LIN {X 0,Y 488.78,Z 301.595,A -85,B 0,C 180,E1 22660.647,E2 22660.647} C_VEL
LIN {X 0,Y 488.836,Z 301.585,A -85,B 0,C 180,E1 22657.258,E2 22657.258} C_VEL
LIN {X 0,Y 488.792,Z 301.599,A -85,B 0,C 180,E1 22653.779,E2 22653.779} C_VEL
LIN {X 0,Y 488.782,Z 301.597,A -85,B 0,C 180,E1 22650.328,E2 22650.328} C_VEL
LIN {X 0,Y 488.822,Z 301.594,A -85,B 0,C 180,E1 22646.898,E2 22646.898} C_VEL
LIN {X 0,Y 488.826,Z 301.564,A -85,B 0,C 180,E1 22643.301,E2 22643.301} C_VEL
LIN {X 0,Y 488.793,Z 301.59,A -85,B 0,C 180,E1 22639.883,E2 22639.883} C_VEL
LIN {X 0,Y 488.796,Z 301.598,A -85,B 0,C 180,E1 22636.225,E2 22636.225} C_VEL
LIN {X 0,Y 488.826,Z 301.575,A -85,B 0,C 180,E1 22632.751,E2 22632.751} C_VEL
LIN {X 0,Y 488.839,Z 301.65,A -85,B 0,C 180,E1 22631.1,E2 22631.1} C_VEL
LIN {X 0,Y 489.193,Z 303.151,A -85,B 0,C 180,E1 22630.866,E2 22630.866} C_VEL
LIN {X 0,Y 497.247,Z 321.838,A -85,B 0,C 180,E1 22628.815,E2 22628.815} C_VEL
LIN {X 0,Y 502.538,Z 335.639,A -85,B 0,C 180,E1 22627.431,E2 22627.431} C_VEL
LIN {X 0,Y 500.242,Z 388.267,A -85,B 0,C 180,E1 22624.007,E2 22624.007} C_VEL
LIN {X 0,Y 502.743,Z 409.204,A -85,B 0,C 180,E1 22623.487,E2 22623.487} C_VEL
LIN {X 0,Y 499.827,Z 627.706,A -85,B 0,C 180,E1 22620.075,E2 22620.075} C_VEL
LIN {X 0,Y 499.277,Z 655.552,A -85,B 0,C 180,E1 22619.579,E2 22619.579} C_VEL
LIN {X 0,Y 498.434,Z 677.22,A -85,B 0,C 180,E1 22618.977,E2 22618.977} C_VEL
LIN {X 0,Y 497.483,Z 697.861,A -85,B 0,C 180,E1 22618.184,E2 22618.184} C_VEL
LIN {X 0,Y 496.413,Z 717.588,A -85,B 0,C 180,E1 22617.207,E2 22617.207} C_VEL
LIN {X 0,Y 495.194,Z 737.474,A -85,B 0,C 180,E1 22615.985,E2 22615.985} C_VEL
LIN {X 0,Y 493.989,Z 756.462,A -85,B 0,C 180,E1 22614.565,E2 22614.565} C_VEL
LIN {X 0,Y 492.797,Z 774.049,A -85,B 0,C 180,E1 22612.989,E2 22612.989} C_VEL
LIN {X 0,Y 491.739,Z 789.65,A -85,B 0,C 180,E1 22611.343,E2 22611.343} C_VEL
LIN {X 0,Y 490.759,Z 804.438,A -85,B 0,C 180,E1 22609.519,E2 22609.519} C_VEL
LIN {X 0,Y 490.048,Z 815.118,A -85,B 0,C 180,E1 22607.944,E2 22607.944} C_VEL
LIN {X 0,Y 489.28,Z 826.646,A -85,B 0,C 180,E1 22605.892,E2 22605.892} C_VEL
LIN {X 0,Y 488.709,Z 836.846,A -85,B 0,C 180,E1 22603.728,E2 22603.728} C_VEL
LIN {X 0,Y 488.31,Z 845.655,A -85,B 0,C 180,E1 22601.456,E2 22601.456} C_VEL
LIN {X 0,Y 488.088,Z 852.685,A -85,B 0,C 180,E1 22599.194,E2 22599.194} C_VEL
LIN {X 0,Y 487.97,Z 858.26,A -85,B 0,C 180,E1 22596.825,E2 22596.825} C_VEL
LIN {X 0,Y 487.913,Z 862.087,A -85,B 0,C 180,E1 22594.466,E2 22594.466} C_VEL
LIN {X 0,Y 487.908,Z 864.304,A -85,B 0,C 180,E1 22592.114,E2 22592.114} C_VEL
LIN {X 0,Y 487.906,Z 864.962,A -85,B 0,C 180,E1 22589.765,E2 22589.765} C_VEL
LIN {X 0,Y 487.905,Z 864.03,A -85,B 0,C 180,E1 22587.416,E2 22587.416} C_VEL
LIN {X 0,Y 487.929,Z 861.446,A -85,B 0,C 180,E1 22585.063,E2 22585.063} C_VEL
LIN {X 0,Y 487.987,Z 857.244,A -85,B 0,C 180,E1 22582.702,E2 22582.702} C_VEL
LIN {X 0,Y 488.126,Z 851.326,A -85,B 0,C 180,E1 22580.331,E2 22580.331} C_VEL
LIN {X 0,Y 488.381,Z 844.01,A -85,B 0,C 180,E1 22578.067,E2 22578.067} C_VEL
LIN {X 0,Y 488.823,Z 834.789,A -85,B 0,C 180,E1 22575.792,E2 22575.792} C_VEL
LIN {X 0,Y 489.44,Z 824.106,A -85,B 0,C 180,E1 22573.626,E2 22573.626} C_VEL
LIN {X 0,Y 490.253,Z 812.019,A -85,B 0,C 180,E1 22571.572,E2 22571.572} C_VEL
LIN {X 0,Y 491.025,Z 800.468,A -85,B 0,C 180,E1 22569.954,E2 22569.954} C_VEL
LIN {X 0,Y 492.085,Z 784.784,A -85,B 0,C 180,E1 22568.109,E2 22568.109} C_VEL
LIN {X 0,Y 493.241,Z 767.415,A -85,B 0,C 180,E1 22566.385,E2 22566.385} C_VEL
LIN {X 0,Y 494.4,Z 750.145,A -85,B 0,C 180,E1 22564.94,E2 22564.94} C_VEL
LIN {X 0,Y 495.552,Z 731.825,A -85,B 0,C 180,E1 22563.649,E2 22563.649} C_VEL
LIN {X 0,Y 496.728,Z 711.811,A -85,B 0,C 180,E1 22562.487,E2 22562.487} C_VEL
LIN {X 0,Y 497.765,Z 692.146,A -85,B 0,C 180,E1 22561.572,E2 22561.572} C_VEL
LIN {X 0,Y 498.696,Z 671.504,A -85,B 0,C 180,E1 22560.837,E2 22560.837} C_VEL
LIN {X 0,Y 499.453,Z 649.882,A -85,B 0,C 180,E1 22560.293,E2 22560.293} C_VEL
LIN {X 0,Y 502.656,Z 414.695,A -85,B 0,C 180,E1 22556.6,E2 22556.6} C_VEL
LIN {X 0,Y 502.523,Z 405.875,A -85,B 0,C 180,E1 22556.443,E2 22556.443} C_VEL
LIN {X 0,Y 500.189,Z 387.515,A -85,B 0,C 180,E1 22555.965,E2 22555.965} C_VEL
LIN {X 0,Y 502.552,Z 335.273,A -85,B 0,C 180,E1 22552.545,E2 22552.545} C_VEL
LIN {X 0,Y 494.184,Z 314.542,A -85,B 0,C 180,E1 22550.409,E2 22550.409} C_VEL
LIN {X 0,Y 488.897,Z 302.02,A -85,B 0,C 180,E1 22548.995,E2 22548.995} C_VEL
LIN {X 0,Y 488.827,Z 301.588,A -85,B 0,C 180,E1 22548.648,E2 22548.648} C_VEL
LIN {X 0,Y 488.832,Z 301.584,A -85,B 0,C 180,E1 22545.049,E2 22545.049} C_VEL
LIN {X 0,Y 488.802,Z 301.566,A -85,B 0,C 180,E1 22541.51,E2 22541.51} C_VEL
LIN {X 0,Y 488.79,Z 301.592,A -85,B 0,C 180,E1 22538.004,E2 22538.004} C_VEL
LIN {X 0,Y 488.813,Z 301.58,A -85,B 0,C 180,E1 22534.482,E2 22534.482} C_VEL
LIN {X 0,Y 488.834,Z 301.587,A -85,B 0,C 180,E1 22530.89,E2 22530.89} C_VEL
LIN {X 0,Y 488.79,Z 301.591,A -85,B 0,C 180,E1 22527.403,E2 22527.403} C_VEL
LIN {X 0,Y 488.779,Z 301.593,A -85,B 0,C 180,E1 22523.884,E2 22523.884} C_VEL
LIN {X 0,Y 488.816,Z 301.598,A -85,B 0,C 180,E1 22520.473,E2 22520.473} C_VEL
LIN {X 0,Y 488.801,Z 301.592,A -85,B 0,C 180,E1 22517.008,E2 22517.008} C_VEL
LIN {X 0,Y 488.765,Z 301.585,A -85,B 0,C 180,E1 22513.606,E2 22513.606} C_VEL
LIN {X 0,Y 488.783,Z 301.596,A -85,B 0,C 180,E1 22510.132,E2 22510.132} C_VEL
LIN {X 0,Y 488.827,Z 301.591,A -85,B 0,C 180,E1 22506.577,E2 22506.577} C_VEL
LIN {X 0,Y 488.77,Z 301.59,A -85,B 0,C 180,E1 22503.049,E2 22503.049} C_VEL
LIN {X 0,Y 488.753,Z 301.6,A -85,B 0,C 180,E1 22499.648,E2 22499.648} C_VEL
LIN {X 0,Y 488.794,Z 301.59,A -85,B 0,C 180,E1 22496.247,E2 22496.247} C_VEL
LIN {X 0,Y 488.783,Z 301.599,A -85,B 0,C 180,E1 22492.79,E2 22492.79} C_VEL
LIN {X 0,Y 488.756,Z 301.598,A -85,B 0,C 180,E1 22489.39,E2 22489.39} C_VEL
LIN {X 0,Y 488.783,Z 301.585,A -85,B 0,C 180,E1 22485.911,E2 22485.911} C_VEL
LIN {X 0,Y 488.808,Z 301.6,A -85,B 0,C 180,E1 22482.501,E2 22482.501} C_VEL
LIN {X 0,Y 488.771,Z 301.593,A -85,B 0,C 180,E1 22479.023,E2 22479.023} C_VEL
LIN {X 0,Y 488.775,Z 301.586,A -85,B 0,C 180,E1 22475.464,E2 22475.464} C_VEL
LIN {X 0,Y 488.83,Z 301.592,A -85,B 0,C 180,E1 22472.069,E2 22472.069} C_VEL
LIN {X 0,Y 488.806,Z 301.597,A -85,B 0,C 180,E1 22468.534,E2 22468.534} C_VEL
LIN {X 0,Y 488.781,Z 301.595,A -85,B 0,C 180,E1 22465.056,E2 22465.056} C_VEL
LIN {X 0,Y 488.801,Z 301.594,A -85,B 0,C 180,E1 22461.549,E2 22461.549} C_VEL
LIN {X 0,Y 488.832,Z 301.59,A -85,B 0,C 180,E1 22458.022,E2 22458.022} C_VEL
LIN {X 0,Y 488.81,Z 301.571,A -85,B 0,C 180,E1 22454.448,E2 22454.448} C_VEL
LIN {X 0,Y 488.793,Z 301.6,A -85,B 0,C 180,E1 22450.887,E2 22450.887} C_VEL
LIN {X 0,Y 488.804,Z 301.585,A -85,B 0,C 180,E1 22447.277,E2 22447.277} C_VEL
LIN {X 0,Y 488.829,Z 301.571,A -85,B 0,C 180,E1 22443.803,E2 22443.803} C_VEL
LIN {X 0,Y 488.825,Z 301.575,A -85,B 0,C 180,E1 22443.535,E2 22443.535} C_VEL
LIN {X 0,Y 488.707,Z 302.659,A -85,B 0,C 180,E1 22443.028,E2 22443.028} C_VEL
LIN {X 0,Y 488.366,Z 306.029,A -85,B 0,C 180,E1 22442.479,E2 22442.479} C_VEL
LIN {X 0,Y 487.643,Z 319.511,A -85,B 0,C 180,E1 22441.022,E2 22441.022} C_VEL
LIN {X 0,Y 488.549,Z 324.711,A -85,B 0,C 180,E1 22440.361,E2 22440.361} C_VEL
LIN {X 0,Y 490.865,Z 331.872,A -85,B 0,C 180,E1 22439.399,E2 22439.399} C_VEL
LIN {X 0,Y 490.606,Z 339.583,A -85,B 0,C 180,E1 22438.658,E2 22438.658} C_VEL
LIN {X 0,Y 494.065,Z 356.306,A -85,B 0,C 180,E1 22438.141,E2 22438.141} C_VEL
LIN {X 0,Y 492.291,Z 551.901,A -85,B 0,C 180,E1 22435.29,E2 22435.29} C_VEL
LIN {X 0,Y 491.896,Z 570.892,A -85,B 0,C 180,E1 22434.786,E2 22434.786} C_VEL
LIN {X 0,Y 491.192,Z 588.904,A -85,B 0,C 180,E1 22434.087,E2 22434.087} C_VEL
LIN {X 0,Y 490.248,Z 606.351,A -85,B 0,C 180,E1 22433.179,E2 22433.179} C_VEL
LIN {X 0,Y 489.098,Z 622.756,A -85,B 0,C 180,E1 22432.095,E2 22432.095} C_VEL
LIN {X 0,Y 487.851,Z 638.101,A -85,B 0,C 180,E1 22430.839,E2 22430.839} C_VEL
LIN {X 0,Y 486.5,Z 652.717,A -85,B 0,C 180,E1 22429.379,E2 22429.379} C_VEL
LIN {X 0,Y 485.184,Z 666.107,A -85,B 0,C 180,E1 22427.757,E2 22427.757} C_VEL
LIN {X 0,Y 483.924,Z 678.429,A -85,B 0,C 180,E1 22425.949,E2 22425.949} C_VEL
LIN {X 0,Y 482.864,Z 689.222,A -85,B 0,C 180,E1 22424.02,E2 22424.02} C_VEL
LIN {X 0,Y 481.974,Z 698.544,A -85,B 0,C 180,E1 22421.973,E2 22421.973} C_VEL
LIN {X 0,Y 481.314,Z 706.381,A -85,B 0,C 180,E1 22419.807,E2 22419.807} C_VEL
LIN {X 0,Y 480.863,Z 712.699,A -85,B 0,C 180,E1 22417.527,E2 22417.527} C_VEL
LIN {X 0,Y 480.577,Z 717.234,A -85,B 0,C 180,E1 22415.252,E2 22415.252} C_VEL
LIN {X 0,Y 480.428,Z 720.208,A -85,B 0,C 180,E1 22412.863,E2 22412.863} C_VEL
LIN {X 0,Y 480.381,Z 721.437,A -85,B 0,C 180,E1 22410.477,E2 22410.477} C_VEL
LIN {X 0,Y 480.403,Z 720.959,A -85,B 0,C 180,E1 22408.092,E2 22408.092} C_VEL
LIN {X 0,Y 480.492,Z 718.906,A -85,B 0,C 180,E1 22405.824,E2 22405.824} C_VEL
LIN {X 0,Y 480.694,Z 715.237,A -85,B 0,C 180,E1 22403.551,E2 22403.551} C_VEL
LIN {X 0,Y 481.06,Z 709.851,A -85,B 0,C 180,E1 22401.273,E2 22401.273} C_VEL
LIN {X 0,Y 481.58,Z 703.016,A -85,B 0,C 180,E1 22399.11,E2 22399.11} C_VEL
LIN {X 0,Y 482.32,Z 694.791,A -85,B 0,C 180,E1 22397.063,E2 22397.063} C_VEL
LIN {X 0,Y 483.286,Z 684.793,A -85,B 0,C 180,E1 22395.054,E2 22395.054} C_VEL
LIN {X 0,Y 484.416,Z 673.543,A -85,B 0,C 180,E1 22393.204,E2 22393.204} C_VEL
LIN {X 0,Y 485.68,Z 661.12,A -85,B 0,C 180,E1 22391.517,E2 22391.517} C_VEL
LIN {X 0,Y 487.013,Z 647.199,A -85,B 0,C 180,E1 22389.95,E2 22389.95} C_VEL
LIN {X 0,Y 488.338,Z 632.237,A -85,B 0,C 180,E1 22388.564,E2 22388.564} C_VEL
LIN {X 0,Y 489.56,Z 616.352,A -85,B 0,C 180,E1 22387.364,E2 22387.364} C_VEL
LIN {X 0,Y 490.6,Z 600.329,A -85,B 0,C 180,E1 22386.393,E2 22386.393} C_VEL
LIN {X 0,Y 491.444,Z 583.063,A -85,B 0,C 180,E1 22385.575,E2 22385.575} C_VEL
LIN {X 0,Y 492.049,Z 564.71,A -85,B 0,C 180,E1 22384.938,E2 22384.938} C_VEL
LIN {X 0,Y 492.337,Z 545.999,A -85,B 0,C 180,E1 22384.513,E2 22384.513} C_VEL
LIN {X 0,Y 493.96,Z 354.759,A -85,B 0,C 180,E1 22381.732,E2 22381.732} C_VEL
LIN {X 0,Y 490.529,Z 338.771,A -85,B 0,C 180,E1 22381.202,E2 22381.202} C_VEL
LIN {X 0,Y 490.727,Z 331.435,A -85,B 0,C 180,E1 22380.458,E2 22380.458} C_VEL
LIN {X 0,Y 484.023,Z 311.463,A -85,B 0,C 180,E1 22377.66,E2 22377.66} C_VEL
LIN {X 0,Y 480.917,Z 302.763,A -85,B 0,C 180,E1 22376.336,E2 22376.336} C_VEL
LIN {X 0,Y 480.867,Z 302.575,A -85,B 0,C 180,E1 22372.767,E2 22372.767} C_VEL
LIN {X 0,Y 480.863,Z 302.589,A -85,B 0,C 180,E1 22369.189,E2 22369.189} C_VEL
LIN {X 0,Y 480.883,Z 302.553,A -85,B 0,C 180,E1 22365.664,E2 22365.664} C_VEL
LIN {X 0,Y 480.895,Z 302.58,A -85,B 0,C 180,E1 22362.028,E2 22362.028} C_VEL
LIN {X 0,Y 480.867,Z 302.582,A -85,B 0,C 180,E1 22358.441,E2 22358.441} C_VEL
LIN {X 0,Y 480.848,Z 302.582,A -85,B 0,C 180,E1 22354.878,E2 22354.878} C_VEL
LIN {X 0,Y 480.86,Z 302.585,A -85,B 0,C 180,E1 22351.288,E2 22351.288} C_VEL
LIN {X 0,Y 480.894,Z 302.581,A -85,B 0,C 180,E1 22347.758,E2 22347.758} C_VEL
LIN {X 0,Y 480.86,Z 302.573,A -85,B 0,C 180,E1 22344.182,E2 22344.182} C_VEL
LIN {X 0,Y 480.835,Z 302.581,A -85,B 0,C 180,E1 22340.657,E2 22340.657} C_VEL
LIN {X 0,Y 480.84,Z 302.588,A -85,B 0,C 180,E1 22337.05,E2 22337.05} C_VEL
LIN {X 0,Y 480.885,Z 302.571,A -85,B 0,C 180,E1 22333.589,E2 22333.589} C_VEL
LIN {X 0,Y 480.844,Z 302.586,A -85,B 0,C 180,E1 22330.06,E2 22330.06} C_VEL
LIN {X 0,Y 480.818,Z 302.588,A -85,B 0,C 180,E1 22326.568,E2 22326.568} C_VEL
LIN {X 0,Y 480.836,Z 302.574,A -85,B 0,C 180,E1 22323.099,E2 22323.099} C_VEL
LIN {X 0,Y 480.876,Z 302.585,A -85,B 0,C 180,E1 22319.524,E2 22319.524} C_VEL
LIN {X 0,Y 480.831,Z 302.58,A -85,B 0,C 180,E1 22315.946,E2 22315.946} C_VEL
LIN {X 0,Y 480.818,Z 302.579,A -85,B 0,C 180,E1 22312.472,E2 22312.472} C_VEL
LIN {X 0,Y 480.845,Z 302.587,A -85,B 0,C 180,E1 22308.943,E2 22308.943} C_VEL
LIN {X 0,Y 480.886,Z 302.576,A -85,B 0,C 180,E1 22305.429,E2 22305.429} C_VEL
LIN {X 0,Y 480.839,Z 302.581,A -85,B 0,C 180,E1 22301.951,E2 22301.951} C_VEL
LIN {X 0,Y 480.834,Z 302.586,A -85,B 0,C 180,E1 22298.353,E2 22298.353} C_VEL
LIN {X 0,Y 480.87,Z 302.585,A -85,B 0,C 180,E1 22294.902,E2 22294.902} C_VEL
LIN {X 0,Y 480.897,Z 302.584,A -85,B 0,C 180,E1 22291.296,E2 22291.296} C_VEL
LIN {X 0,Y 480.853,Z 302.585,A -85,B 0,C 180,E1 22287.808,E2 22287.808} C_VEL
LIN {X 0,Y 480.845,Z 302.554,A -85,B 0,C 180,E1 22284.187,E2 22284.187} C_VEL
LIN {X 0,Y 480.874,Z 302.584,A -85,B 0,C 180,E1 22280.642,E2 22280.642} C_VEL
LIN {X 0,Y 480.892,Z 302.564,A -85,B 0,C 180,E1 22277.041,E2 22277.041} C_VEL
LIN {X 0,Y 480.874,Z 302.557,A -85,B 0,C 180,E1 22273.477,E2 22273.477} C_VEL
LIN {X 0,Y 480.906,Z 302.863,A -85,B 0,C 180,E1 22271.68,E2 22271.68} C_VEL
LIN {X 0,Y 483.793,Z 309.643,A -85,B 0,C 180,E1 22270.851,E2 22270.851} C_VEL
LIN {X 0,Y 493.151,Z 332.06,A -85,B 0,C 180,E1 22268.407,E2 22268.407} C_VEL
LIN {X 0,Y 495.521,Z 338.509,A -85,B 0,C 180,E1 22267.762,E2 22267.762} C_VEL
LIN {X 0,Y 493.157,Z 387.828,A -85,B 0,C 180,E1 22264.503,E2 22264.503} C_VEL
LIN {X 0,Y 495.787,Z 410.337,A -85,B 0,C 180,E1 22263.929,E2 22263.929} C_VEL
LIN {X 0,Y 492.138,Z 649.298,A -85,B 0,C 180,E1 22260.091,E2 22260.091} C_VEL
LIN {X 0,Y 491.304,Z 671.237,A -85,B 0,C 180,E1 22259.525,E2 22259.525} C_VEL
LIN {X 0,Y 490.246,Z 692.612,A -85,B 0,C 180,E1 22258.74,E2 22258.74} C_VEL
LIN {X 0,Y 489.065,Z 713.265,A -85,B 0,C 180,E1 22257.746,E2 22257.746} C_VEL
LIN {X 0,Y 487.862,Z 732.316,A -85,B 0,C 180,E1 22256.602,E2 22256.602} C_VEL
LIN {X 0,Y 486.592,Z 751.078,A -85,B 0,C 180,E1 22255.237,E2 22255.237} C_VEL
LIN {X 0,Y 485.262,Z 769.522,A -85,B 0,C 180,E1 22253.625,E2 22253.625} C_VEL
LIN {X 0,Y 484.067,Z 786.361,A -85,B 0,C 180,E1 22251.874,E2 22251.874} C_VEL
LIN {X 0,Y 483.041,Z 800.956,A -85,B 0,C 180,E1 22250.096,E2 22250.096} C_VEL
LIN {X 0,Y 482.123,Z 814.745,A -85,B 0,C 180,E1 22248.124,E2 22248.124} C_VEL
LIN {X 0,Y 481.36,Z 827.01,A -85,B 0,C 180,E1 22246.037,E2 22246.037} C_VEL
LIN {X 0,Y 480.828,Z 836.331,A -85,B 0,C 180,E1 22244.081,E2 22244.081} C_VEL
LIN {X 0,Y 480.378,Z 845.25,A -85,B 0,C 180,E1 22241.769,E2 22241.769} C_VEL
LIN {X 0,Y 480.123,Z 852.375,A -85,B 0,C 180,E1 22239.469,E2 22239.469} C_VEL
LIN {X 0,Y 479.983,Z 858.006,A -85,B 0,C 180,E1 22237.059,E2 22237.059} C_VEL
LIN {X 0,Y 479.919,Z 861.926,A -85,B 0,C 180,E1 22234.66,E2 22234.66} C_VEL
LIN {X 0,Y 479.907,Z 864.303,A -85,B 0,C 180,E1 22232.149,E2 22232.149} C_VEL
LIN {X 0,Y 479.906,Z 864.962,A -85,B 0,C 180,E1 22229.761,E2 22229.761} C_VEL
LIN {X 0,Y 479.907,Z 864.03,A -85,B 0,C 180,E1 22227.373,E2 22227.373} C_VEL
LIN {X 0,Y 479.931,Z 861.445,A -85,B 0,C 180,E1 22224.98,E2 22224.98} C_VEL
LIN {X 0,Y 479.994,Z 857.159,A -85,B 0,C 180,E1 22222.54,E2 22222.54} C_VEL
LIN {X 0,Y 480.146,Z 851.326,A -85,B 0,C 180,E1 22220.168,E2 22220.168} C_VEL
LIN {X 0,Y 480.431,Z 844.009,A -85,B 0,C 180,E1 22217.866,E2 22217.866} C_VEL
LIN {X 0,Y 480.919,Z 834.786,A -85,B 0,C 180,E1 22215.553,E2 22215.553} C_VEL
LIN {X 0,Y 481.435,Z 825.653,A -85,B 0,C 180,E1 22213.718,E2 22213.718} C_VEL
LIN {X 0,Y 482.226,Z 813.101,A -85,B 0,C 180,E1 22211.63,E2 22211.63} C_VEL
LIN {X 0,Y 483.169,Z 799.084,A -85,B 0,C 180,E1 22209.657,E2 22209.657} C_VEL
LIN {X 0,Y 484.324,Z 782.977,A -85,B 0,C 180,E1 22207.741,E2 22207.741} C_VEL
LIN {X 0,Y 485.559,Z 765.638,A -85,B 0,C 180,E1 22206.004,E2 22206.004} C_VEL
LIN {X 0,Y 486.861,Z 747.174,A -85,B 0,C 180,E1 22204.452,E2 22204.452} C_VEL
LIN {X 0,Y 488.045,Z 729.442,A -85,B 0,C 180,E1 22203.211,E2 22203.211} C_VEL
LIN {X 0,Y 489.249,Z 710.207,A -85,B 0,C 180,E1 22202.096,E2 22202.096} C_VEL
LIN {X 0,Y 490.344,Z 690.339,A -85,B 0,C 180,E1 22201.169,E2 22201.169} C_VEL
LIN {X 0,Y 491.367,Z 669.669,A -85,B 0,C 180,E1 22200.429,E2 22200.429} C_VEL
LIN {X 0,Y 492.173,Z 648.273,A -85,B 0,C 180,E1 22199.887,E2 22199.887} C_VEL
LIN {X 0,Y 495.806,Z 409.537,A -85,B 0,C 180,E1 22196.057,E2 22196.057} C_VEL
LIN {X 0,Y 493.099,Z 386.873,A -85,B 0,C 180,E1 22195.46,E2 22195.46} C_VEL
LIN {X 0,Y 495.495,Z 338.18,A -85,B 0,C 180,E1 22192.214,E2 22192.214} C_VEL
LIN {X 0,Y 486.73,Z 316.473,A -85,B 0,C 180,E1 22189.925,E2 22189.925} C_VEL
LIN {X 0,Y 480.947,Z 303.081,A -85,B 0,C 180,E1 22188.366,E2 22188.366} C_VEL
LIN {X 0,Y 480.86,Z 302.587,A -85,B 0,C 180,E1 22188.107,E2 22188.107} C_VEL
LIN {X 0,Y 480.875,Z 302.584,A -85,B 0,C 180,E1 22184.483,E2 22184.483} C_VEL
LIN {X 0,Y 480.898,Z 302.556,A -85,B 0,C 180,E1 22180.818,E2 22180.818} C_VEL
LIN {X 0,Y 480.878,Z 302.561,A -85,B 0,C 180,E1 22177.22,E2 22177.22} C_VEL
LIN {X 0,Y 480.849,Z 302.585,A -85,B 0,C 180,E1 22173.724,E2 22173.724} C_VEL
LIN {X 0,Y 480.851,Z 302.589,A -85,B 0,C 180,E1 22170.074,E2 22170.074} C_VEL
LIN {X 0,Y 480.887,Z 302.578,A -85,B 0,C 180,E1 22166.616,E2 22166.616} C_VEL
LIN {X 0,Y 480.875,Z 302.576,A -85,B 0,C 180,E1 22163.01,E2 22163.01} C_VEL
LIN {X 0,Y 480.835,Z 302.584,A -85,B 0,C 180,E1 22159.559,E2 22159.559} C_VEL
LIN {X 0,Y 480.836,Z 302.588,A -85,B 0,C 180,E1 22155.931,E2 22155.931} C_VEL
LIN {X 0,Y 480.877,Z 302.576,A -85,B 0,C 180,E1 22152.488,E2 22152.488} C_VEL
LIN {X 0,Y 480.849,Z 302.58,A -85,B 0,C 180,E1 22148.972,E2 22148.972} C_VEL
LIN {X 0,Y 480.818,Z 302.589,A -85,B 0,C 180,E1 22145.489,E2 22145.489} C_VEL
LIN {X 0,Y 480.827,Z 302.584,A -85,B 0,C 180,E1 22141.906,E2 22141.906} C_VEL
LIN {X 0,Y 480.87,Z 302.579,A -85,B 0,C 180,E1 22138.451,E2 22138.451} C_VEL
LIN {X 0,Y 480.836,Z 302.586,A -85,B 0,C 180,E1 22134.87,E2 22134.87} C_VEL
LIN {X 0,Y 480.813,Z 302.574,A -85,B 0,C 180,E1 22131.389,E2 22131.389} C_VEL
LIN {X 0,Y 480.838,Z 302.586,A -85,B 0,C 180,E1 22127.876,E2 22127.876} C_VEL
LIN {X 0,Y 480.878,Z 302.577,A -85,B 0,C 180,E1 22124.441,E2 22124.441} C_VEL
LIN {X 0,Y 480.834,Z 302.582,A -85,B 0,C 180,E1 22120.945,E2 22120.945} C_VEL
LIN {X 0,Y 480.831,Z 302.587,A -85,B 0,C 180,E1 22117.375,E2 22117.375} C_VEL
LIN {X 0,Y 480.865,Z 302.585,A -85,B 0,C 180,E1 22113.844,E2 22113.844} C_VEL
LIN {X 0,Y 480.886,Z 302.575,A -85,B 0,C 180,E1 22110.34,E2 22110.34} C_VEL
LIN {X 0,Y 480.846,Z 302.586,A -85,B 0,C 180,E1 22106.847,E2 22106.847} C_VEL
LIN {X 0,Y 480.846,Z 302.586,A -85,B 0,C 180,E1 22103.181,E2 22103.181} C_VEL
LIN {X 0,Y 480.878,Z 302.582,A -85,B 0,C 180,E1 22099.711,E2 22099.711} C_VEL
LIN {X 0,Y 480.89,Z 302.58,A -85,B 0,C 180,E1 22096.175,E2 22096.175} C_VEL
LIN {X 0,Y 480.861,Z 302.567,A -85,B 0,C 180,E1 22092.601,E2 22092.601} C_VEL
LIN {X 0,Y 480.853,Z 302.564,A -85,B 0,C 180,E1 22089.052,E2 22089.052} C_VEL
LIN {X 0,Y 480.878,Z 302.572,A -85,B 0,C 180,E1 22085.457,E2 22085.457} C_VEL
LIN {X 0,Y 480.921,Z 302.801,A -85,B 0,C 180,E1 22083.554,E2 22083.554} C_VEL
LIN {X 0,Y 487.772,Z 322.317,A -85,B 0,C 180,E1 22080.69,E2 22080.69} C_VEL
LIN {X 0,Y 488.549,Z 324.711,A -85,B 0,C 180,E1 22080.361,E2 22080.361} C_VEL
LIN {X 0,Y 488.628,Z 327.991,A -85,B 0,C 180,E1 22079.994,E2 22079.994} C_VEL
LIN {X 0,Y 486.858,Z 333.513,A -85,B 0,C 180,E1 22079.555,E2 22079.555} C_VEL
LIN {X 0,Y 484.726,Z 340.308,A -85,B 0,C 180,E1 22079.192,E2 22079.192} C_VEL
LIN {X 0,Y 484.615,Z 344.653,A -85,B 0,C 180,E1 22079.02,E2 22079.02} C_VEL
LIN {X 0,Y 484.753,Z 345.376,A -85,B 0,C 180,E1 22078.995,E2 22078.995} C_VEL
LIN {X 0,Y 487.233,Z 357.819,A -85,B 0,C 180,E1 22078.611,E2 22078.611} C_VEL
LIN {X 0,Y 485.291,Z 552.929,A -85,B 0,C 180,E1 22075.73,E2 22075.73} C_VEL
LIN {X 0,Y 484.868,Z 571.912,A -85,B 0,C 180,E1 22075.219,E2 22075.219} C_VEL
LIN {X 0,Y 484.142,Z 589.615,A -85,B 0,C 180,E1 22074.525,E2 22074.525} C_VEL
LIN {X 0,Y 483.129,Z 607.284,A -85,B 0,C 180,E1 22073.597,E2 22073.597} C_VEL
LIN {X 0,Y 481.92,Z 623.618,A -85,B 0,C 180,E1 22072.506,E2 22072.506} C_VEL
LIN {X 0,Y 480.579,Z 639.115,A -85,B 0,C 180,E1 22071.223,E2 22071.223} C_VEL
LIN {X 0,Y 479.096,Z 654.161,A -85,B 0,C 180,E1 22069.696,E2 22069.696} C_VEL
LIN {X 0,Y 477.689,Z 667.548,A -85,B 0,C 180,E1 22068.046,E2 22068.046} C_VEL
LIN {X 0,Y 476.342,Z 679.831,A -85,B 0,C 180,E1 22066.21,E2 22066.21} C_VEL
LIN {X 0,Y 475.201,Z 690.591,A -85,B 0,C 180,E1 22064.251,E2 22064.251} C_VEL
LIN {X 0,Y 474.239,Z 699.883,A -85,B 0,C 180,E1 22062.171,E2 22062.171} C_VEL
LIN {X 0,Y 473.519,Z 707.693,A -85,B 0,C 180,E1 22059.971,E2 22059.971} C_VEL
LIN {X 0,Y 473.043,Z 713.704,A -85,B 0,C 180,E1 22057.774,E2 22057.774} C_VEL
LIN {X 0,Y 472.713,Z 718.291,A -85,B 0,C 180,E1 22055.462,E2 22055.462} C_VEL
LIN {X 0,Y 472.54,Z 721.219,A -85,B 0,C 180,E1 22053.154,E2 22053.154} C_VEL
LIN {X 0,Y 472.479,Z 722.598,A -85,B 0,C 180,E1 22050.728,E2 22050.728} C_VEL
LIN {X 0,Y 472.492,Z 722.289,A -85,B 0,C 180,E1 22048.302,E2 22048.302} C_VEL
LIN {X 0,Y 472.593,Z 720.28,A -85,B 0,C 180,E1 22045.875,E2 22045.875} C_VEL
LIN {X 0,Y 472.831,Z 716.498,A -85,B 0,C 180,E1 22043.443,E2 22043.443} C_VEL
LIN {X 0,Y 473.239,Z 711.145,A -85,B 0,C 180,E1 22041.128,E2 22041.128} C_VEL
LIN {X 0,Y 473.829,Z 704.179,A -85,B 0,C 180,E1 22038.882,E2 22038.882} C_VEL
LIN {X 0,Y 474.676,Z 695.612,A -85,B 0,C 180,E1 22036.727,E2 22036.727} C_VEL
LIN {X 0,Y 475.696,Z 685.842,A -85,B 0,C 180,E1 22034.747,E2 22034.747} C_VEL
LIN {X 0,Y 476.872,Z 674.958,A -85,B 0,C 180,E1 22032.931,E2 22032.931} C_VEL
LIN {X 0,Y 478.22,Z 662.576,A -85,B 0,C 180,E1 22031.218,E2 22031.218} C_VEL
LIN {X 0,Y 479.641,Z 648.71,A -85,B 0,C 180,E1 22029.628,E2 22029.628} C_VEL
LIN {X 0,Y 481.046,Z 633.823,A -85,B 0,C 180,E1 22028.223,E2 22028.223} C_VEL
LIN {X 0,Y 482.358,Z 617.867,A -85,B 0,C 180,E1 22026.994,E2 22026.994} C_VEL
LIN {X 0,Y 483.516,Z 601.071,A -85,B 0,C 180,E1 22025.961,E2 22025.961} C_VEL
LIN {X 0,Y 484.412,Z 583.702,A -85,B 0,C 180,E1 22025.131,E2 22025.131} C_VEL
LIN {X 0,Y 485.046,Z 565.341,A -85,B 0,C 180,E1 22024.49,E2 22024.49} C_VEL
LIN {X 0,Y 485.345,Z 546.648,A -85,B 0,C 180,E1 22024.064,E2 22024.064} C_VEL
LIN {X 0,Y 487.126,Z 356.194,A -85,B 0,C 180,E1 22021.259,E2 22021.259} C_VEL
LIN {X 0,Y 483.5,Z 339.269,A -85,B 0,C 180,E1 22020.687,E2 22020.687} C_VEL
LIN {X 0,Y 483.498,Z 334.249,A -85,B 0,C 180,E1 22020.171,E2 22020.171} C_VEL
LIN {X 0,Y 477.178,Z 315.408,A -85,B 0,C 180,E1 22017.499,E2 22017.499} C_VEL
LIN {X 0,Y 472.986,Z 303.82,A -85,B 0,C 180,E1 22015.72,E2 22015.72} C_VEL
LIN {X 0,Y 472.934,Z 303.576,A -85,B 0,C 180,E1 22013.403,E2 22013.403} C_VEL
LIN {X 0,Y 472.955,Z 303.563,A -85,B 0,C 180,E1 22009.746,E2 22009.746} C_VEL
LIN {X 0,Y 472.95,Z 303.537,A -85,B 0,C 180,E1 22006.1,E2 22006.1} C_VEL
LIN {X 0,Y 472.933,Z 303.573,A -85,B 0,C 180,E1 22002.454,E2 22002.454} C_VEL
LIN {X 0,Y 472.912,Z 303.573,A -85,B 0,C 180,E1 21998.898,E2 21998.898} C_VEL
LIN {X 0,Y 472.92,Z 303.573,A -85,B 0,C 180,E1 21995.253,E2 21995.253} C_VEL
LIN {X 0,Y 472.95,Z 303.576,A -85,B 0,C 180,E1 21991.621,E2 21991.621} C_VEL
LIN {X 0,Y 472.947,Z 303.568,A -85,B 0,C 180,E1 21987.991,E2 21987.991} C_VEL
LIN {X 0,Y 472.903,Z 303.562,A -85,B 0,C 180,E1 21984.482,E2 21984.482} C_VEL
LIN {X 0,Y 472.897,Z 303.57,A -85,B 0,C 180,E1 21980.852,E2 21980.852} C_VEL
LIN {X 0,Y 472.923,Z 303.577,A -85,B 0,C 180,E1 21977.344,E2 21977.344} C_VEL
LIN {X 0,Y 472.935,Z 303.558,A -85,B 0,C 180,E1 21973.822,E2 21973.822} C_VEL
LIN {X 0,Y 472.888,Z 303.575,A -85,B 0,C 180,E1 21970.354,E2 21970.354} C_VEL
LIN {X 0,Y 472.88,Z 303.577,A -85,B 0,C 180,E1 21966.678,E2 21966.678} C_VEL
LIN {X 0,Y 472.901,Z 303.562,A -85,B 0,C 180,E1 21963.152,E2 21963.152} C_VEL
LIN {X 0,Y 472.933,Z 303.575,A -85,B 0,C 180,E1 21959.555,E2 21959.555} C_VEL
LIN {X 0,Y 472.888,Z 303.569,A -85,B 0,C 180,E1 21955.999,E2 21955.999} C_VEL
LIN {X 0,Y 472.879,Z 303.568,A -85,B 0,C 180,E1 21952.467,E2 21952.467} C_VEL
LIN {X 0,Y 472.904,Z 303.576,A -85,B 0,C 180,E1 21948.907,E2 21948.907} C_VEL
LIN {X 0,Y 472.951,Z 303.566,A -85,B 0,C 180,E1 21945.304,E2 21945.304} C_VEL
LIN {X 0,Y 472.92,Z 303.565,A -85,B 0,C 180,E1 21941.67,E2 21941.67} C_VEL
LIN {X 0,Y 472.897,Z 303.575,A -85,B 0,C 180,E1 21938.15,E2 21938.15} C_VEL
LIN {X 0,Y 472.903,Z 303.575,A -85,B 0,C 180,E1 21934.449,E2 21934.449} C_VEL
LIN {X 0,Y 472.939,Z 303.574,A -85,B 0,C 180,E1 21930.906,E2 21930.906} C_VEL
LIN {X 0,Y 472.952,Z 303.576,A -85,B 0,C 180,E1 21927.286,E2 21927.286} C_VEL
LIN {X 0,Y 472.918,Z 303.538,A -85,B 0,C 180,E1 21923.702,E2 21923.702} C_VEL
LIN {X 0,Y 472.913,Z 303.572,A -85,B 0,C 180,E1 21920.126,E2 21920.126} C_VEL
LIN {X 0,Y 472.936,Z 303.564,A -85,B 0,C 180,E1 21916.599,E2 21916.599} C_VEL
LIN {X 0,Y 472.952,Z 303.545,A -85,B 0,C 180,E1 21912.99,E2 21912.99} C_VEL
LIN {X 0,Y 472.971,Z 303.857,A -85,B 0,C 180,E1 21912.351,E2 21912.351} C_VEL
LIN {X 0,Y 474.297,Z 307.162,A -85,B 0,C 180,E1 21911.914,E2 21911.914} C_VEL
LIN {X 0,Y 483.1,Z 327.539,A -85,B 0,C 180,E1 21909.561,E2 21909.561} C_VEL
LIN {X 0,Y 488.516,Z 341.444,A -85,B 0,C 180,E1 21908.097,E2 21908.097} C_VEL
LIN {X 0,Y 486.114,Z 387.432,A -85,B 0,C 180,E1 21905.012,E2 21905.012} C_VEL
LIN {X 0,Y 488.878,Z 411.471,A -85,B 0,C 180,E1 21904.387,E2 21904.387} C_VEL
LIN {X 0,Y 484.865,Z 648.353,A -85,B 0,C 180,E1 21900.495,E2 21900.495} C_VEL
LIN {X 0,Y 483.955,Z 670.357,A -85,B 0,C 180,E1 21899.916,E2 21899.916} C_VEL
LIN {X 0,Y 482.806,Z 691.638,A -85,B 0,C 180,E1 21899.121,E2 21899.121} C_VEL
LIN {X 0,Y 481.561,Z 712.103,A -85,B 0,C 180,E1 21898.119,E2 21898.119} C_VEL
LIN {X 0,Y 480.295,Z 730.708,A -85,B 0,C 180,E1 21896.988,E2 21896.988} C_VEL
LIN {X 0,Y 478.924,Z 749.74,A -85,B 0,C 180,E1 21895.592,E2 21895.592} C_VEL
LIN {X 0,Y 477.537,Z 768.213,A -85,B 0,C 180,E1 21893.965,E2 21893.965} C_VEL
LIN {X 0,Y 476.367,Z 783.896,A -85,B 0,C 180,E1 21892.327,E2 21892.327} C_VEL
LIN {X 0,Y 475.213,Z 799.277,A -85,B 0,C 180,E1 21890.442,E2 21890.442} C_VEL
LIN {X 0,Y 474.238,Z 813.225,A -85,B 0,C 180,E1 21888.422,E2 21888.422} C_VEL
LIN {X 0,Y 473.441,Z 825.496,A -85,B 0,C 180,E1 21886.312,E2 21886.312} C_VEL
LIN {X 0,Y 472.854,Z 835.853,A -85,B 0,C 180,E1 21884.198,E2 21884.198} C_VEL
LIN {X 0,Y 472.411,Z 844.926,A -85,B 0,C 180,E1 21881.971,E2 21881.971} C_VEL
LIN {X 0,Y 472.167,Z 851.3,A -85,B 0,C 180,E1 21879.999,E2 21879.999} C_VEL
LIN {X 0,Y 472.01,Z 856.987,A -85,B 0,C 180,E1 21877.669,E2 21877.669} C_VEL
LIN {X 0,Y 471.933,Z 861.287,A -85,B 0,C 180,E1 21875.227,E2 21875.227} C_VEL
LIN {X 0,Y 471.912,Z 863.954,A -85,B 0,C 180,E1 21872.793,E2 21872.793} C_VEL
LIN {X 0,Y 471.902,Z 864.939,A -85,B 0,C 180,E1 21870.364,E2 21870.364} C_VEL
LIN {X 0,Y 471.908,Z 864.37,A -85,B 0,C 180,E1 21867.936,E2 21867.936} C_VEL
LIN {X 0,Y 471.914,Z 862.243,A -85,B 0,C 180,E1 21865.504,E2 21865.504} C_VEL
LIN {X 0,Y 471.981,Z 858.51,A -85,B 0,C 180,E1 21863.065,E2 21863.065} C_VEL
LIN {X 0,Y 472.12,Z 852.991,A -85,B 0,C 180,E1 21860.615,E2 21860.615} C_VEL
LIN {X 0,Y 472.336,Z 846.662,A -85,B 0,C 180,E1 21858.523,E2 21858.523} C_VEL
LIN {X 0,Y 472.733,Z 838.068,A -85,B 0,C 180,E1 21856.298,E2 21856.298} C_VEL
LIN {X 0,Y 473.329,Z 827.515,A -85,B 0,C 180,E1 21854.062,E2 21854.062} C_VEL
LIN {X 0,Y 474.086,Z 815.458,A -85,B 0,C 180,E1 21851.94,E2 21851.94} C_VEL
LIN {X 0,Y 475.017,Z 802.008,A -85,B 0,C 180,E1 21849.935,E2 21849.935} C_VEL
LIN {X 0,Y 476.154,Z 786.614,A -85,B 0,C 180,E1 21847.987,E2 21847.987} C_VEL
LIN {X 0,Y 477.371,Z 770.423,A -85,B 0,C 180,E1 21846.248,E2 21846.248} C_VEL
LIN {X 0,Y 478.663,Z 753.619,A -85,B 0,C 180,E1 21844.719,E2 21844.719} C_VEL
LIN {X 0,Y 480.034,Z 734.524,A -85,B 0,C 180,E1 21843.263,E2 21843.263} C_VEL
LIN {X 0,Y 481.407,Z 714.406,A -85,B 0,C 180,E1 21842.006,E2 21842.006} C_VEL
LIN {X 0,Y 482.647,Z 694.418,A -85,B 0,C 180,E1 21841.004,E2 21841.004} C_VEL
LIN {X 0,Y 483.736,Z 674.042,A -85,B 0,C 180,E1 21840.21,E2 21840.21} C_VEL
LIN {X 0,Y 484.691,Z 652.903,A -85,B 0,C 180,E1 21839.611,E2 21839.611} C_VEL
LIN {X 0,Y 485.301,Z 625.97,A -85,B 0,C 180,E1 21839.119,E2 21839.119} C_VEL
LIN {X 0,Y 488.876,Z 409.615,A -85,B 0,C 180,E1 21835.579,E2 21835.579} C_VEL
LIN {X 0,Y 486.051,Z 386.321,A -85,B 0,C 180,E1 21834.944,E2 21834.944} C_VEL
LIN {X 0,Y 488.478,Z 341.211,A -85,B 0,C 180,E1 21831.885,E2 21831.885} C_VEL
LIN {X 0,Y 479.993,Z 320.207,A -85,B 0,C 180,E1 21829.623,E2 21829.623} C_VEL
LIN {X 0,Y 473.78,Z 306.31,A -85,B 0,C 180,E1 21827.975,E2 21827.975} C_VEL
LIN {X 0,Y 472.959,Z 303.774,A -85,B 0,C 180,E1 21827.625,E2 21827.625} C_VEL
LIN {X 0,Y 472.919,Z 303.578,A -85,B 0,C 180,E1 21824.073,E2 21824.073} C_VEL
LIN {X 0,Y 472.932,Z 303.554,A -85,B 0,C 180,E1 21820.441,E2 21820.441} C_VEL
LIN {X 0,Y 472.954,Z 303.54,A -85,B 0,C 180,E1 21816.898,E2 21816.898} C_VEL
LIN {X 0,Y 472.926,Z 303.572,A -85,B 0,C 180,E1 21813.346,E2 21813.346} C_VEL
LIN {X 0,Y 472.905,Z 303.577,A -85,B 0,C 180,E1 21809.792,E2 21809.792} C_VEL
LIN {X 0,Y 472.916,Z 303.575,A -85,B 0,C 180,E1 21806.223,E2 21806.223} C_VEL
LIN {X 0,Y 472.954,Z 303.563,A -85,B 0,C 180,E1 21802.629,E2 21802.629} C_VEL
LIN {X 0,Y 472.927,Z 303.567,A -85,B 0,C 180,E1 21799.001,E2 21799.001} C_VEL
LIN {X 0,Y 472.893,Z 303.576,A -85,B 0,C 180,E1 21795.45,E2 21795.45} C_VEL
LIN {X 0,Y 472.889,Z 303.576,A -85,B 0,C 180,E1 21791.785,E2 21791.785} C_VEL
LIN {X 0,Y 472.917,Z 303.563,A -85,B 0,C 180,E1 21788.266,E2 21788.266} C_VEL
LIN {X 0,Y 472.914,Z 303.577,A -85,B 0,C 180,E1 21784.851,E2 21784.851} C_VEL
LIN {X 0,Y 472.877,Z 303.573,A -85,B 0,C 180,E1 21781.332,E2 21781.332} C_VEL
LIN {X 0,Y 472.874,Z 303.566,A -85,B 0,C 180,E1 21777.697,E2 21777.697} C_VEL
LIN {X 0,Y 472.916,Z 303.577,A -85,B 0,C 180,E1 21774.175,E2 21774.175} C_VEL
LIN {X 0,Y 472.903,Z 303.561,A -85,B 0,C 180,E1 21770.753,E2 21770.753} C_VEL
LIN {X 0,Y 472.881,Z 303.575,A -85,B 0,C 180,E1 21767.297,E2 21767.297} C_VEL
LIN {X 0,Y 472.898,Z 303.576,A -85,B 0,C 180,E1 21763.714,E2 21763.714} C_VEL
LIN {X 0,Y 472.942,Z 303.56,A -85,B 0,C 180,E1 21760.179,E2 21760.179} C_VEL
LIN {X 0,Y 472.912,Z 303.577,A -85,B 0,C 180,E1 21756.711,E2 21756.711} C_VEL
LIN {X 0,Y 472.897,Z 303.576,A -85,B 0,C 180,E1 21753.153,E2 21753.153} C_VEL
LIN {X 0,Y 472.914,Z 303.572,A -85,B 0,C 180,E1 21749.608,E2 21749.608} C_VEL
LIN {X 0,Y 472.953,Z 303.563,A -85,B 0,C 180,E1 21746.074,E2 21746.074} C_VEL
LIN {X 0,Y 472.934,Z 303.568,A -85,B 0,C 180,E1 21742.447,E2 21742.447} C_VEL
LIN {X 0,Y 472.908,Z 303.573,A -85,B 0,C 180,E1 21739.006,E2 21739.006} C_VEL
LIN {X 0,Y 472.925,Z 303.565,A -85,B 0,C 180,E1 21735.419,E2 21735.419} C_VEL
LIN {X 0,Y 472.955,Z 303.563,A -85,B 0,C 180,E1 21731.913,E2 21731.913} C_VEL
LIN {X 0,Y 472.944,Z 303.544,A -85,B 0,C 180,E1 21728.274,E2 21728.274} C_VEL
LIN {X 0,Y 472.921,Z 303.549,A -85,B 0,C 180,E1 21724.66,E2 21724.66} C_VEL
LIN {X 0,Y 472.989,Z 303.849,A -85,B 0,C 180,E1 21724.174,E2 21724.174} C_VEL
LIN {X 0,Y 479.913,Z 323.35,A -85,B 0,C 180,E1 21721.249,E2 21721.249} C_VEL
LIN {X 0,Y 483.686,Z 335.439,A -85,B 0,C 180,E1 21719.606,E2 21719.606} C_VEL
LIN {X 0,Y 483.581,Z 340.099,A -85,B 0,C 180,E1 21719.172,E2 21719.172} C_VEL
LIN {X 0,Y 484.753,Z 345.376,A -85,B 0,C 180,E1 21718.995,E2 21718.995} C_VEL
LIN {X 0,Y 485.299,Z 350.755,A -85,B 0,C 180,E1 21718.868,E2 21718.868} C_VEL
LIN {X 0,Y 484.453,Z 358.492,A -85,B 0,C 180,E1 21718.806,E2 21718.806} C_VEL
LIN {X 0,Y 480.505,Z 376.325,A -85,B 0,C 180,E1 21718.815,E2 21718.815} C_VEL
LIN {X 0,Y 480.145,Z 380.86,A -85,B 0,C 180,E1 21718.769,E2 21718.769} C_VEL
LIN {X 0,Y 478.317,Z 553.703,A -85,B 0,C 180,E1 21716.188,E2 21716.188} C_VEL
LIN {X 0,Y 477.869,Z 572.764,A -85,B 0,C 180,E1 21715.669,E2 21715.669} C_VEL
LIN {X 0,Y 477.113,Z 590.257,A -85,B 0,C 180,E1 21714.977,E2 21714.977} C_VEL
LIN {X 0,Y 476.054,Z 607.893,A -85,B 0,C 180,E1 21714.045,E2 21714.045} C_VEL
LIN {X 0,Y 474.761,Z 624.43,A -85,B 0,C 180,E1 21712.93,E2 21712.93} C_VEL
LIN {X 0,Y 473.266,Z 640.634,A -85,B 0,C 180,E1 21711.567,E2 21711.567} C_VEL
LIN {X 0,Y 471.754,Z 655.085,A -85,B 0,C 180,E1 21710.081,E2 21710.081} C_VEL
LIN {X 0,Y 470.309,Z 668.075,A -85,B 0,C 180,E1 21708.467,E2 21708.467} C_VEL
LIN {X 0,Y 468.853,Z 680.476,A -85,B 0,C 180,E1 21706.604,E2 21706.604} C_VEL
LIN {X 0,Y 467.611,Z 691.334,A -85,B 0,C 180,E1 21704.614,E2 21704.614} C_VEL
LIN {X 0,Y 466.559,Z 700.713,A -85,B 0,C 180,E1 21702.5,E2 21702.5} C_VEL
LIN {X 0,Y 465.758,Z 708.599,A -85,B 0,C 180,E1 21700.263,E2 21700.263} C_VEL
LIN {X 0,Y 465.198,Z 714.956,A -85,B 0,C 180,E1 21697.906,E2 21697.906} C_VEL
LIN {X 0,Y 464.835,Z 719.52,A -85,B 0,C 180,E1 21695.554,E2 21695.554} C_VEL
LIN {X 0,Y 464.636,Z 722.483,A -85,B 0,C 180,E1 21693.143,E2 21693.143} C_VEL
LIN {X 0,Y 464.57,Z 723.8,A -85,B 0,C 180,E1 21690.74,E2 21690.74} C_VEL
LIN {X 0,Y 464.586,Z 723.493,A -85,B 0,C 180,E1 21688.273,E2 21688.273} C_VEL
LIN {X 0,Y 464.7,Z 721.497,A -85,B 0,C 180,E1 21685.805,E2 21685.805} C_VEL
LIN {X 0,Y 464.967,Z 717.736,A -85,B 0,C 180,E1 21683.332,E2 21683.332} C_VEL
LIN {X 0,Y 465.414,Z 712.406,A -85,B 0,C 180,E1 21680.977,E2 21680.977} C_VEL
LIN {X 0,Y 466.043,Z 705.625,A -85,B 0,C 180,E1 21678.742,E2 21678.742} C_VEL
LIN {X 0,Y 466.915,Z 697.454,A -85,B 0,C 180,E1 21676.628,E2 21676.628} C_VEL
LIN {X 0,Y 467.983,Z 687.949,A -85,B 0,C 180,E1 21674.638,E2 21674.638} C_VEL
LIN {X 0,Y 469.237,Z 677.125,A -85,B 0,C 180,E1 21672.772,E2 21672.772} C_VEL
LIN {X 0,Y 470.736,Z 664.265,A -85,B 0,C 180,E1 21670.944,E2 21670.944} C_VEL
LIN {X 0,Y 472.276,Z 650.183,A -85,B 0,C 180,E1 21669.296,E2 21669.296} C_VEL
LIN {X 0,Y 473.722,Z 635.791,A -85,B 0,C 180,E1 21667.907,E2 21667.907} C_VEL
LIN {X 0,Y 475.147,Z 619.6,A -85,B 0,C 180,E1 21666.631,E2 21666.631} C_VEL
LIN {X 0,Y 476.381,Z 602.871,A -85,B 0,C 180,E1 21665.577,E2 21665.577} C_VEL
LIN {X 0,Y 477.366,Z 585.014,A -85,B 0,C 180,E1 21664.705,E2 21664.705} C_VEL
LIN {X 0,Y 478.047,Z 566.621,A -85,B 0,C 180,E1 21664.051,E2 21664.051} C_VEL
LIN {X 0,Y 478.371,Z 547.772,A -85,B 0,C 180,E1 21663.611,E2 21663.611} C_VEL
LIN {X 0,Y 480.338,Z 357.695,A -85,B 0,C 180,E1 21660.775,E2 21660.775} C_VEL
LIN {X 0,Y 476.501,Z 339.597,A -85,B 0,C 180,E1 21660.144,E2 21660.144} C_VEL
LIN {X 0,Y 476.305,Z 337.122,A -85,B 0,C 180,E1 21659.868,E2 21659.868} C_VEL
LIN {X 0,Y 469.867,Z 318.049,A -85,B 0,C 180,E1 21657.138,E2 21657.138} C_VEL
LIN {X 0,Y 465.02,Z 304.778,A -85,B 0,C 180,E1 21655.041,E2 21655.041} C_VEL
LIN {X 0,Y 464.991,Z 304.532,A -85,B 0,C 180,E1 21651.423,E2 21651.423} C_VEL
LIN {X 0,Y 465.012,Z 304.548,A -85,B 0,C 180,E1 21647.868,E2 21647.868} C_VEL
LIN {X 0,Y 465.011,Z 304.552,A -85,B 0,C 180,E1 21644.16,E2 21644.16} C_VEL
LIN {X 0,Y 464.981,Z 304.56,A -85,B 0,C 180,E1 21640.62,E2 21640.62} C_VEL
LIN {X 0,Y 464.975,Z 304.563,A -85,B 0,C 180,E1 21637.021,E2 21637.021} C_VEL
LIN {X 0,Y 464.991,Z 304.555,A -85,B 0,C 180,E1 21633.4,E2 21633.4} C_VEL
LIN {X 0,Y 465.02,Z 304.55,A -85,B 0,C 180,E1 21629.781,E2 21629.781} C_VEL
LIN {X 0,Y 464.988,Z 304.563,A -85,B 0,C 180,E1 21626.156,E2 21626.156} C_VEL
LIN {X 0,Y 464.959,Z 304.565,A -85,B 0,C 180,E1 21622.639,E2 21622.639} C_VEL
LIN {X 0,Y 464.957,Z 304.557,A -85,B 0,C 180,E1 21618.949,E2 21618.949} C_VEL
LIN {X 0,Y 464.996,Z 304.553,A -85,B 0,C 180,E1 21615.464,E2 21615.464} C_VEL
LIN {X 0,Y 464.981,Z 304.562,A -85,B 0,C 180,E1 21611.914,E2 21611.914} C_VEL
LIN {X 0,Y 464.943,Z 304.549,A -85,B 0,C 180,E1 21608.409,E2 21608.409} C_VEL
LIN {X 0,Y 464.94,Z 304.564,A -85,B 0,C 180,E1 21604.688,E2 21604.688} C_VEL
LIN {X 0,Y 464.959,Z 304.567,A -85,B 0,C 180,E1 21601.109,E2 21601.109} C_VEL
LIN {X 0,Y 464.978,Z 304.55,A -85,B 0,C 180,E1 21597.659,E2 21597.659} C_VEL
LIN {X 0,Y 464.95,Z 304.566,A -85,B 0,C 180,E1 21594.075,E2 21594.075} C_VEL
LIN {X 0,Y 464.944,Z 304.562,A -85,B 0,C 180,E1 21590.469,E2 21590.469} C_VEL
LIN {X 0,Y 464.969,Z 304.549,A -85,B 0,C 180,E1 21586.929,E2 21586.929} C_VEL
LIN {X 0,Y 465.006,Z 304.561,A -85,B 0,C 180,E1 21583.383,E2 21583.383} C_VEL
LIN {X 0,Y 464.976,Z 304.563,A -85,B 0,C 180,E1 21579.745,E2 21579.745} C_VEL
LIN {X 0,Y 464.959,Z 304.558,A -85,B 0,C 180,E1 21576.289,E2 21576.289} C_VEL
LIN {X 0,Y 464.982,Z 304.554,A -85,B 0,C 180,E1 21572.741,E2 21572.741} C_VEL
LIN {X 0,Y 465.019,Z 304.552,A -85,B 0,C 180,E1 21569.221,E2 21569.221} C_VEL
LIN {X 0,Y 464.989,Z 304.544,A -85,B 0,C 180,E1 21565.562,E2 21565.562} C_VEL
LIN {X 0,Y 464.972,Z 304.556,A -85,B 0,C 180,E1 21562.048,E2 21562.048} C_VEL
LIN {X 0,Y 464.982,Z 304.528,A -85,B 0,C 180,E1 21558.442,E2 21558.442} C_VEL
LIN {X 0,Y 465.01,Z 304.541,A -85,B 0,C 180,E1 21554.801,E2 21554.801} C_VEL
LIN {X 0,Y 465.044,Z 304.759,A -85,B 0,C 180,E1 21553.079,E2 21553.079} C_VEL
LIN {X 0,Y 465.721,Z 306.981,A -85,B 0,C 180,E1 21552.757,E2 21552.757} C_VEL
LIN {X 0,Y 472.984,Z 323.119,A -85,B 0,C 180,E1 21550.782,E2 21550.782} C_VEL
LIN {X 0,Y 481.5,Z 344.299,A -85,B 0,C 180,E1 21548.449,E2 21548.449} C_VEL
LIN {X 0,Y 479.097,Z 386.938,A -85,B 0,C 180,E1 21545.539,E2 21545.539} C_VEL
LIN {X 0,Y 482.005,Z 412.581,A -85,B 0,C 180,E1 21544.859,E2 21544.859} C_VEL
LIN {X 0,Y 477.723,Z 644.596,A -85,B 0,C 180,E1 21540.972,E2 21540.972} C_VEL
LIN {X 0,Y 476.799,Z 665.677,A -85,B 0,C 180,E1 21540.435,E2 21540.435} C_VEL
LIN {X 0,Y 475.665,Z 685.998,A -85,B 0,C 180,E1 21539.705,E2 21539.705} C_VEL
LIN {X 0,Y 474.346,Z 706.844,A -85,B 0,C 180,E1 21538.723,E2 21538.723} C_VEL
LIN {X 0,Y 472.963,Z 726.232,A -85,B 0,C 180,E1 21537.578,E2 21537.578} C_VEL
LIN {X 0,Y 471.573,Z 744.752,A -85,B 0,C 180,E1 21536.251,E2 21536.251} C_VEL
LIN {X 0,Y 470.153,Z 762.824,A -85,B 0,C 180,E1 21534.701,E2 21534.701} C_VEL
LIN {X 0,Y 468.751,Z 780.33,A -85,B 0,C 180,E1 21532.909,E2 21532.909} C_VEL
LIN {X 0,Y 467.508,Z 796.111,A -85,B 0,C 180,E1 21530.991,E2 21530.991} C_VEL
LIN {X 0,Y 466.494,Z 809.868,A -85,B 0,C 180,E1 21529.013,E2 21529.013} C_VEL
LIN {X 0,Y 465.62,Z 822.611,A -85,B 0,C 180,E1 21526.851,E2 21526.851} C_VEL
LIN {X 0,Y 464.958,Z 833.863,A -85,B 0,C 180,E1 21524.572,E2 21524.572} C_VEL
LIN {X 0,Y 464.481,Z 843.122,A -85,B 0,C 180,E1 21522.304,E2 21522.304} C_VEL
LIN {X 0,Y 464.185,Z 850.907,A -85,B 0,C 180,E1 21519.922,E2 21519.922} C_VEL
LIN {X 0,Y 464.011,Z 856.844,A -85,B 0,C 180,E1 21517.553,E2 21517.553} C_VEL
LIN {X 0,Y 463.935,Z 861.3,A -85,B 0,C 180,E1 21515.069,E2 21515.069} C_VEL
LIN {X 0,Y 463.91,Z 863.893,A -85,B 0,C 180,E1 21512.718,E2 21512.718} C_VEL
LIN {X 0,Y 463.906,Z 864.873,A -85,B 0,C 180,E1 21510.247,E2 21510.247} C_VEL
LIN {X 0,Y 463.908,Z 864.253,A -85,B 0,C 180,E1 21507.9,E2 21507.9} C_VEL
LIN {X 0,Y 463.915,Z 862.156,A -85,B 0,C 180,E1 21505.55,E2 21505.55} C_VEL
LIN {X 0,Y 463.98,Z 858.403,A -85,B 0,C 180,E1 21503.193,E2 21503.193} C_VEL
LIN {X 0,Y 464.119,Z 852.952,A -85,B 0,C 180,E1 21500.827,E2 21500.827} C_VEL
LIN {X 0,Y 464.376,Z 845.677,A -85,B 0,C 180,E1 21498.426,E2 21498.426} C_VEL
LIN {X 0,Y 464.799,Z 836.645,A -85,B 0,C 180,E1 21496.059,E2 21496.059} C_VEL
LIN {X 0,Y 465.407,Z 826.027,A -85,B 0,C 180,E1 21493.783,E2 21493.783} C_VEL
LIN {X 0,Y 466.262,Z 813.125,A -85,B 0,C 180,E1 21491.496,E2 21491.496} C_VEL
LIN {X 0,Y 467.257,Z 799.418,A -85,B 0,C 180,E1 21489.456,E2 21489.456} C_VEL
LIN {X 0,Y 468.448,Z 784.198,A -85,B 0,C 180,E1 21487.539,E2 21487.539} C_VEL
LIN {X 0,Y 469.768,Z 767.411,A -85,B 0,C 180,E1 21485.747,E2 21485.747} C_VEL
LIN {X 0,Y 471.24,Z 748.867,A -85,B 0,C 180,E1 21484.083,E2 21484.083} C_VEL
LIN {X 0,Y 472.683,Z 730.027,A -85,B 0,C 180,E1 21482.675,E2 21482.675} C_VEL
LIN {X 0,Y 474.109,Z 710.405,A -85,B 0,C 180,E1 21481.468,E2 21481.468} C_VEL
LIN {X 0,Y 475.395,Z 690.615,A -85,B 0,C 180,E1 21480.484,E2 21480.484} C_VEL
LIN {X 0,Y 476.663,Z 668.946,A -85,B 0,C 180,E1 21479.663,E2 21479.663} C_VEL
LIN {X 0,Y 477.657,Z 646.844,A -85,B 0,C 180,E1 21479.072,E2 21479.072} C_VEL
LIN {X 0,Y 481.919,Z 417.222,A -85,B 0,C 180,E1 21475.218,E2 21475.218} C_VEL
LIN {X 0,Y 481.796,Z 409.235,A -85,B 0,C 180,E1 21475.065,E2 21475.065} C_VEL
LIN {X 0,Y 479.031,Z 385.93,A -85,B 0,C 180,E1 21474.422,E2 21474.422} C_VEL
LIN {X 0,Y 481.428,Z 344.114,A -85,B 0,C 180,E1 21471.534,E2 21471.534} C_VEL
LIN {X 0,Y 472.656,Z 322.365,A -85,B 0,C 180,E1 21469.135,E2 21469.135} C_VEL
LIN {X 0,Y 465.083,Z 304.995,A -85,B 0,C 180,E1 21466.989,E2 21466.989} C_VEL
LIN {X 0,Y 465.002,Z 304.531,A -85,B 0,C 180,E1 21466.617,E2 21466.617} C_VEL
LIN {X 0,Y 465.014,Z 304.537,A -85,B 0,C 180,E1 21462.969,E2 21462.969} C_VEL
LIN {X 0,Y 464.996,Z 304.563,A -85,B 0,C 180,E1 21459.37,E2 21459.37} C_VEL
LIN {X 0,Y 464.967,Z 304.528,A -85,B 0,C 180,E1 21455.796,E2 21455.796} C_VEL
LIN {X 0,Y 464.973,Z 304.562,A -85,B 0,C 180,E1 21452.082,E2 21452.082} C_VEL
LIN {X 0,Y 465.004,Z 304.561,A -85,B 0,C 180,E1 21448.512,E2 21448.512} C_VEL
LIN {X 0,Y 465.013,Z 304.565,A -85,B 0,C 180,E1 21444.789,E2 21444.789} C_VEL
LIN {X 0,Y 464.971,Z 304.563,A -85,B 0,C 180,E1 21441.31,E2 21441.31} C_VEL
LIN {X 0,Y 464.954,Z 304.56,A -85,B 0,C 180,E1 21437.708,E2 21437.708} C_VEL
LIN {X 0,Y 464.967,Z 304.551,A -85,B 0,C 180,E1 21434.118,E2 21434.118} C_VEL
LIN {X 0,Y 465,Z 304.564,A -85,B 0,C 180,E1 21430.531,E2 21430.531} C_VEL
LIN {X 0,Y 464.972,Z 304.557,A -85,B 0,C 180,E1 21426.916,E2 21426.916} C_VEL
LIN {X 0,Y 464.939,Z 304.558,A -85,B 0,C 180,E1 21423.452,E2 21423.452} C_VEL
LIN {X 0,Y 464.942,Z 304.567,A -85,B 0,C 180,E1 21419.753,E2 21419.753} C_VEL
LIN {X 0,Y 464.97,Z 304.555,A -85,B 0,C 180,E1 21416.177,E2 21416.177} C_VEL
LIN {X 0,Y 464.984,Z 304.556,A -85,B 0,C 180,E1 21412.587,E2 21412.587} C_VEL
LIN {X 0,Y 464.954,Z 304.565,A -85,B 0,C 180,E1 21408.966,E2 21408.966} C_VEL
LIN {X 0,Y 464.943,Z 304.552,A -85,B 0,C 180,E1 21405.397,E2 21405.397} C_VEL
LIN {X 0,Y 464.97,Z 304.559,A -85,B 0,C 180,E1 21401.832,E2 21401.832} C_VEL
LIN {X 0,Y 465.011,Z 304.564,A -85,B 0,C 180,E1 21398.162,E2 21398.162} C_VEL
LIN {X 0,Y 464.988,Z 304.551,A -85,B 0,C 180,E1 21394.528,E2 21394.528} C_VEL
LIN {X 0,Y 464.961,Z 304.56,A -85,B 0,C 180,E1 21391.063,E2 21391.063} C_VEL
LIN {X 0,Y 464.966,Z 304.563,A -85,B 0,C 180,E1 21387.333,E2 21387.333} C_VEL
LIN {X 0,Y 464.996,Z 304.562,A -85,B 0,C 180,E1 21383.738,E2 21383.738} C_VEL
LIN {X 0,Y 465.021,Z 304.562,A -85,B 0,C 180,E1 21380.137,E2 21380.137} C_VEL
LIN {X 0,Y 464.995,Z 304.564,A -85,B 0,C 180,E1 21376.437,E2 21376.437} C_VEL
LIN {X 0,Y 464.975,Z 304.537,A -85,B 0,C 180,E1 21372.804,E2 21372.804} C_VEL
LIN {X 0,Y 464.977,Z 304.538,A -85,B 0,C 180,E1 21369.079,E2 21369.079} C_VEL
LIN {X 0,Y 464.998,Z 304.545,A -85,B 0,C 180,E1 21365.418,E2 21365.418} C_VEL
LIN {X 0,Y 465.022,Z 304.832,A -85,B 0,C 180,E1 21364.843,E2 21364.843} C_VEL
LIN {X 0,Y 471.654,Z 323.172,A -85,B 0,C 180,E1 21362.009,E2 21362.009} C_VEL
LIN {X 0,Y 476.557,Z 338.304,A -85,B 0,C 180,E1 21359.893,E2 21359.893} C_VEL
LIN {X 0,Y 476.607,Z 340.692,A -85,B 0,C 180,E1 21359.699,E2 21359.699} C_VEL
LIN {X 0,Y 480.435,Z 359.218,A -85,B 0,C 180,E1 21359.096,E2 21359.096} C_VEL
LIN {X 0,Y 480.145,Z 380.86,A -85,B 0,C 180,E1 21358.769,E2 21358.769} C_VEL
LIN {X 0,Y 479.198,Z 388.556,A -85,B 0,C 180,E1 21358.717,E2 21358.717} C_VEL
LIN {X 0,Y 473.655,Z 409.052,A -85,B 0,C 180,E1 21358.807,E2 21358.807} C_VEL
LIN {X 0,Y 472.928,Z 415.659,A -85,B 0,C 180,E1 21358.756,E2 21358.756} C_VEL
LIN {X 0,Y 471.37,Z 554.407,A -85,B 0,C 180,E1 21356.659,E2 21356.659} C_VEL
LIN {X 0,Y 470.896,Z 573.572,A -85,B 0,C 180,E1 21356.132,E2 21356.132} C_VEL
LIN {X 0,Y 470.073,Z 591.528,A -85,B 0,C 180,E1 21355.411,E2 21355.411} C_VEL
LIN {X 0,Y 468.963,Z 608.953,A -85,B 0,C 180,E1 21354.475,E2 21354.475} C_VEL
LIN {X 0,Y 467.544,Z 626.01,A -85,B 0,C 180,E1 21353.304,E2 21353.304} C_VEL
LIN {X 0,Y 466.037,Z 641.481,A -85,B 0,C 180,E1 21351.985,E2 21351.985} C_VEL
LIN {X 0,Y 464.431,Z 655.983,A -85,B 0,C 180,E1 21350.477,E2 21350.477} C_VEL
LIN {X 0,Y 462.834,Z 669.456,A -85,B 0,C 180,E1 21348.776,E2 21348.776} C_VEL
LIN {X 0,Y 461.286,Z 681.817,A -85,B 0,C 180,E1 21346.884,E2 21346.884} C_VEL
LIN {X 0,Y 459.958,Z 692.644,A -85,B 0,C 180,E1 21344.863,E2 21344.863} C_VEL
LIN {X 0,Y 458.83,Z 701.997,A -85,B 0,C 180,E1 21342.714,E2 21342.714} C_VEL
LIN {X 0,Y 457.962,Z 709.86,A -85,B 0,C 180,E1 21340.44,E2 21340.44} C_VEL
LIN {X 0,Y 457.353,Z 716.195,A -85,B 0,C 180,E1 21338.043,E2 21338.043} C_VEL
LIN {X 0,Y 456.956,Z 720.742,A -85,B 0,C 180,E1 21335.651,E2 21335.651} C_VEL
LIN {X 0,Y 456.74,Z 723.638,A -85,B 0,C 180,E1 21333.263,E2 21333.263} C_VEL
LIN {X 0,Y 456.661,Z 725.002,A -85,B 0,C 180,E1 21330.753,E2 21330.753} C_VEL
LIN {X 0,Y 456.679,Z 724.697,A -85,B 0,C 180,E1 21328.244,E2 21328.244} C_VEL
LIN {X 0,Y 456.807,Z 722.71,A -85,B 0,C 180,E1 21325.732,E2 21325.732} C_VEL
LIN {X 0,Y 457.102,Z 718.964,A -85,B 0,C 180,E1 21323.217,E2 21323.217} C_VEL
LIN {X 0,Y 457.589,Z 713.653,A -85,B 0,C 180,E1 21320.822,E2 21320.822} C_VEL
LIN {X 0,Y 458.275,Z 706.892,A -85,B 0,C 180,E1 21318.549,E2 21318.549} C_VEL
LIN {X 0,Y 459.214,Z 698.747,A -85,B 0,C 180,E1 21316.4,E2 21316.4} C_VEL
LIN {X 0,Y 460.44,Z 688.616,A -85,B 0,C 180,E1 21314.25,E2 21314.25} C_VEL
LIN {X 0,Y 461.863,Z 677.188,A -85,B 0,C 180,E1 21312.276,E2 21312.276} C_VEL
LIN {X 0,Y 463.439,Z 664.431,A -85,B 0,C 180,E1 21310.464,E2 21310.464} C_VEL
LIN {X 0,Y 465.056,Z 650.47,A -85,B 0,C 180,E1 21308.827,E2 21308.827} C_VEL
LIN {X 0,Y 466.65,Z 635.471,A -85,B 0,C 180,E1 21307.382,E2 21307.382} C_VEL
LIN {X 0,Y 468.035,Z 620.346,A -85,B 0,C 180,E1 21306.187,E2 21306.187} C_VEL
LIN {X 0,Y 469.311,Z 603.926,A -85,B 0,C 180,E1 21305.142,E2 21305.142} C_VEL
LIN {X 0,Y 470.343,Z 586.287,A -85,B 0,C 180,E1 21304.267,E2 21304.267} C_VEL
LIN {X 0,Y 471.079,Z 567.644,A -85,B 0,C 180,E1 21303.591,E2 21303.591} C_VEL
LIN {X 0,Y 471.426,Z 548.714,A -85,B 0,C 180,E1 21303.142,E2 21303.142} C_VEL
LIN {X 0,Y 473.554,Z 359.044,A -85,B 0,C 180,E1 21300.271,E2 21300.271} C_VEL
LIN {X 0,Y 469.391,Z 340.655,A -85,B 0,C 180,E1 21299.622,E2 21299.622} C_VEL
LIN {X 0,Y 463.748,Z 323.819,A -85,B 0,C 180,E1 21297.231,E2 21297.231} C_VEL
LIN {X 0,Y 457.853,Z 308.147,A -85,B 0,C 180,E1 21294.76,E2 21294.76} C_VEL
LIN {X 0,Y 457.088,Z 305.664,A -85,B 0,C 180,E1 21294.304,E2 21294.304} C_VEL
LIN {X 0,Y 457.054,Z 305.524,A -85,B 0,C 180,E1 21290.625,E2 21290.625} C_VEL
LIN {X 0,Y 457.04,Z 305.52,A -85,B 0,C 180,E1 21286.958,E2 21286.958} C_VEL
LIN {X 0,Y 457.046,Z 305.555,A -85,B 0,C 180,E1 21283.215,E2 21283.215} C_VEL
LIN {X 0,Y 457.072,Z 305.554,A -85,B 0,C 180,E1 21279.647,E2 21279.647} C_VEL
LIN {X 0,Y 457.077,Z 305.551,A -85,B 0,C 180,E1 21275.892,E2 21275.892} C_VEL
LIN {X 0,Y 457.052,Z 305.549,A -85,B 0,C 180,E1 21272.262,E2 21272.262} C_VEL
LIN {X 0,Y 457.027,Z 305.548,A -85,B 0,C 180,E1 21268.686,E2 21268.686} C_VEL
LIN {X 0,Y 457.025,Z 305.539,A -85,B 0,C 180,E1 21264.976,E2 21264.976} C_VEL
LIN {X 0,Y 457.054,Z 305.549,A -85,B 0,C 180,E1 21261.428,E2 21261.428} C_VEL
LIN {X 0,Y 457.06,Z 305.546,A -85,B 0,C 180,E1 21257.834,E2 21257.834} C_VEL
LIN {X 0,Y 457.019,Z 305.538,A -85,B 0,C 180,E1 21254.267,E2 21254.267} C_VEL
LIN {X 0,Y 457.007,Z 305.553,A -85,B 0,C 180,E1 21250.59,E2 21250.59} C_VEL
LIN {X 0,Y 457.009,Z 305.555,A -85,B 0,C 180,E1 21246.911,E2 21246.911} C_VEL
LIN {X 0,Y 457.043,Z 305.537,A -85,B 0,C 180,E1 21243.387,E2 21243.387} C_VEL
LIN {X 0,Y 457.031,Z 305.556,A -85,B 0,C 180,E1 21239.75,E2 21239.75} C_VEL
LIN {X 0,Y 457.004,Z 305.546,A -85,B 0,C 180,E1 21236.111,E2 21236.111} C_VEL
LIN {X 0,Y 457.002,Z 305.545,A -85,B 0,C 180,E1 21232.457,E2 21232.457} C_VEL
LIN {X 0,Y 457.026,Z 305.554,A -85,B 0,C 180,E1 21228.9,E2 21228.9} C_VEL
LIN {X 0,Y 457.071,Z 305.542,A -85,B 0,C 180,E1 21225.301,E2 21225.301} C_VEL
LIN {X 0,Y 457.044,Z 305.541,A -85,B 0,C 180,E1 21221.638,E2 21221.638} C_VEL
LIN {X 0,Y 457.024,Z 305.553,A -85,B 0,C 180,E1 21218.031,E2 21218.031} C_VEL
LIN {X 0,Y 457.024,Z 305.554,A -85,B 0,C 180,E1 21214.331,E2 21214.331} C_VEL
LIN {X 0,Y 457.052,Z 305.552,A -85,B 0,C 180,E1 21210.79,E2 21210.79} C_VEL
LIN {X 0,Y 457.075,Z 305.551,A -85,B 0,C 180,E1 21207.138,E2 21207.138} C_VEL
LIN {X 0,Y 457.055,Z 305.511,A -85,B 0,C 180,E1 21203.485,E2 21203.485} C_VEL
LIN {X 0,Y 457.036,Z 305.541,A -85,B 0,C 180,E1 21199.967,E2 21199.967} C_VEL
LIN {X 0,Y 457.042,Z 305.553,A -85,B 0,C 180,E1 21196.212,E2 21196.212} C_VEL
LIN {X 0,Y 457.062,Z 305.676,A -85,B 0,C 180,E1 21193.848,E2 21193.848} C_VEL
LIN {X 0,Y 457.472,Z 307.266,A -85,B 0,C 180,E1 21193.57,E2 21193.57} C_VEL
LIN {X 0,Y 462.54,Z 318.305,A -85,B 0,C 180,E1 21192.145,E2 21192.145} C_VEL
LIN {X 0,Y 470.549,Z 337.177,A -85,B 0,C 180,E1 21189.908,E2 21189.908} C_VEL
LIN {X 0,Y 474.52,Z 347.604,A -85,B 0,C 180,E1 21188.774,E2 21188.774} C_VEL
LIN {X 0,Y 472.12,Z 386.495,A -85,B 0,C 180,E1 21186.081,E2 21186.081} C_VEL
LIN {X 0,Y 475.165,Z 413.726,A -85,B 0,C 180,E1 21185.344,E2 21185.344} C_VEL
LIN {X 0,Y 470.643,Z 641.643,A -85,B 0,C 180,E1 21181.463,E2 21181.463} C_VEL
LIN {X 0,Y 469.666,Z 663.065,A -85,B 0,C 180,E1 21180.926,E2 21180.926} C_VEL
LIN {X 0,Y 468.44,Z 683.801,A -85,B 0,C 180,E1 21180.18,E2 21180.18} C_VEL
LIN {X 0,Y 467.029,Z 704.15,A -85,B 0,C 180,E1 21179.216,E2 21179.216} C_VEL
LIN {X 0,Y 465.511,Z 724.195,A -85,B 0,C 180,E1 21178.021,E2 21178.021} C_VEL
LIN {X 0,Y 463.96,Z 743.389,A -85,B 0,C 180,E1 21176.631,E2 21176.631} C_VEL
LIN {X 0,Y 462.458,Z 761.5,A -85,B 0,C 180,E1 21175.056,E2 21175.056} C_VEL
LIN {X 0,Y 460.987,Z 778.905,A -85,B 0,C 180,E1 21173.25,E2 21173.25} C_VEL
LIN {X 0,Y 459.681,Z 794.746,A -85,B 0,C 180,E1 21171.299,E2 21171.299} C_VEL
LIN {X 0,Y 458.601,Z 808.779,A -85,B 0,C 180,E1 21169.259,E2 21169.259} C_VEL
LIN {X 0,Y 457.674,Z 821.782,A -85,B 0,C 180,E1 21167.022,E2 21167.022} C_VEL
LIN {X 0,Y 456.995,Z 832.984,A -85,B 0,C 180,E1 21164.702,E2 21164.702} C_VEL
LIN {X 0,Y 456.51,Z 842.323,A -85,B 0,C 180,E1 21162.356,E2 21162.356} C_VEL
LIN {X 0,Y 456.225,Z 849.97,A -85,B 0,C 180,E1 21159.97,E2 21159.97} C_VEL
LIN {X 0,Y 456.07,Z 855.847,A -85,B 0,C 180,E1 21157.558,E2 21157.558} C_VEL
LIN {X 0,Y 456.011,Z 860.066,A -85,B 0,C 180,E1 21155.158,E2 21155.158} C_VEL
LIN {X 0,Y 455.994,Z 862.711,A -85,B 0,C 180,E1 21152.765,E2 21152.765} C_VEL
LIN {X 0,Y 455.985,Z 863.702,A -85,B 0,C 180,E1 21150.377,E2 21150.377} C_VEL
LIN {X 0,Y 455.989,Z 863.084,A -85,B 0,C 180,E1 21147.864,E2 21147.864} C_VEL
LIN {X 0,Y 455.993,Z 860.931,A -85,B 0,C 180,E1 21145.473,E2 21145.473} C_VEL
LIN {X 0,Y 456.052,Z 857.151,A -85,B 0,C 180,E1 21143.074,E2 21143.074} C_VEL
LIN {X 0,Y 456.182,Z 851.659,A -85,B 0,C 180,E1 21140.666,E2 21140.666} C_VEL
LIN {X 0,Y 456.429,Z 844.406,A -85,B 0,C 180,E1 21138.245,E2 21138.245} C_VEL
LIN {X 0,Y 456.835,Z 835.774,A -85,B 0,C 180,E1 21135.94,E2 21135.94} C_VEL
LIN {X 0,Y 457.454,Z 825.167,A -85,B 0,C 180,E1 21133.623,E2 21133.623} C_VEL
LIN {X 0,Y 458.281,Z 813.035,A -85,B 0,C 180,E1 21131.426,E2 21131.426} C_VEL
LIN {X 0,Y 459.3,Z 799.458,A -85,B 0,C 180,E1 21129.35,E2 21129.35} C_VEL
LIN {X 0,Y 460.592,Z 783.658,A -85,B 0,C 180,E1 21127.308,E2 21127.308} C_VEL
LIN {X 0,Y 462.014,Z 766.602,A -85,B 0,C 180,E1 21125.449,E2 21125.449} C_VEL
LIN {X 0,Y 463.508,Z 748.798,A -85,B 0,C 180,E1 21123.815,E2 21123.815} C_VEL
LIN {X 0,Y 465.015,Z 730.37,A -85,B 0,C 180,E1 21122.397,E2 21122.397} C_VEL
LIN {X 0,Y 466.529,Z 711.204,A -85,B 0,C 180,E1 21121.171,E2 21121.171} C_VEL
LIN {X 0,Y 468.035,Z 689.959,A -85,B 0,C 180,E1 21120.079,E2 21120.079} C_VEL
LIN {X 0,Y 469.413,Z 668.411,A -85,B 0,C 180,E1 21119.239,E2 21119.239} C_VEL
LIN {X 0,Y 470.478,Z 646.724,A -85,B 0,C 180,E1 21118.641,E2 21118.641} C_VEL
LIN {X 0,Y 471.694,Z 588.524,A -85,B 0,C 180,E1 21117.624,E2 21117.624} C_VEL
LIN {X 0,Y 475.091,Z 411.358,A -85,B 0,C 180,E1 21114.607,E2 21114.607} C_VEL
LIN {X 0,Y 472.05,Z 385.383,A -85,B 0,C 180,E1 21113.875,E2 21113.875} C_VEL
LIN {X 0,Y 474.446,Z 347.142,A -85,B 0,C 180,E1 21111.189,E2 21111.189} C_VEL
LIN {X 0,Y 466.077,Z 326.392,A -85,B 0,C 180,E1 21108.85,E2 21108.85} C_VEL
LIN {X 0,Y 458.118,Z 308.607,A -85,B 0,C 180,E1 21106.617,E2 21106.617} C_VEL
LIN {X 0,Y 457.083,Z 305.806,A -85,B 0,C 180,E1 21106.209,E2 21106.209} C_VEL
LIN {X 0,Y 457.043,Z 305.557,A -85,B 0,C 180,E1 21104.149,E2 21104.149} C_VEL
LIN {X 0,Y 457.06,Z 305.526,A -85,B 0,C 180,E1 21100.52,E2 21100.52} C_VEL
LIN {X 0,Y 457.073,Z 305.515,A -85,B 0,C 180,E1 21096.982,E2 21096.982} C_VEL
LIN {X 0,Y 457.051,Z 305.55,A -85,B 0,C 180,E1 21093.305,E2 21093.305} C_VEL
LIN {X 0,Y 457.029,Z 305.555,A -85,B 0,C 180,E1 21089.715,E2 21089.715} C_VEL
LIN {X 0,Y 457.033,Z 305.555,A -85,B 0,C 180,E1 21086.086,E2 21086.086} C_VEL
LIN {X 0,Y 457.062,Z 305.542,A -85,B 0,C 180,E1 21082.509,E2 21082.509} C_VEL
LIN {X 0,Y 457.058,Z 305.541,A -85,B 0,C 180,E1 21078.89,E2 21078.89} C_VEL
LIN {X 0,Y 457.025,Z 305.554,A -85,B 0,C 180,E1 21075.254,E2 21075.254} C_VEL
LIN {X 0,Y 457.01,Z 305.554,A -85,B 0,C 180,E1 21071.612,E2 21071.612} C_VEL
LIN {X 0,Y 457.014,Z 305.542,A -85,B 0,C 180,E1 21067.922,E2 21067.922} C_VEL
LIN {X 0,Y 457.048,Z 305.547,A -85,B 0,C 180,E1 21064.391,E2 21064.391} C_VEL
LIN {X 0,Y 457.051,Z 305.55,A -85,B 0,C 180,E1 21060.626,E2 21060.626} C_VEL
LIN {X 0,Y 457.007,Z 305.539,A -85,B 0,C 180,E1 21056.99,E2 21056.99} C_VEL
LIN {X 0,Y 456.998,Z 305.555,A -85,B 0,C 180,E1 21053.349,E2 21053.349} C_VEL
LIN {X 0,Y 457.008,Z 305.554,A -85,B 0,C 180,E1 21049.665,E2 21049.665} C_VEL
LIN {X 0,Y 457.042,Z 305.536,A -85,B 0,C 180,E1 21046.075,E2 21046.075} C_VEL
LIN {X 0,Y 457.057,Z 305.552,A -85,B 0,C 180,E1 21042.429,E2 21042.429} C_VEL
LIN {X 0,Y 457.025,Z 305.548,A -85,B 0,C 180,E1 21038.839,E2 21038.839} C_VEL
LIN {X 0,Y 457.016,Z 305.539,A -85,B 0,C 180,E1 21035.218,E2 21035.218} C_VEL
LIN {X 0,Y 457.032,Z 305.548,A -85,B 0,C 180,E1 21031.575,E2 21031.575} C_VEL
LIN {X 0,Y 457.074,Z 305.551,A -85,B 0,C 180,E1 21028.036,E2 21028.036} C_VEL
LIN {X 0,Y 457.057,Z 305.553,A -85,B 0,C 180,E1 21024.415,E2 21024.415} C_VEL
LIN {X 0,Y 457.035,Z 305.553,A -85,B 0,C 180,E1 21020.784,E2 21020.784} C_VEL
LIN {X 0,Y 457.036,Z 305.554,A -85,B 0,C 180,E1 21017.127,E2 21017.127} C_VEL
LIN {X 0,Y 457.055,Z 305.514,A -85,B 0,C 180,E1 21013.557,E2 21013.557} C_VEL
LIN {X 0,Y 457.079,Z 305.533,A -85,B 0,C 180,E1 21009.86,E2 21009.86} C_VEL
LIN {X 0,Y 457.07,Z 305.551,A -85,B 0,C 180,E1 21006.176,E2 21006.176} C_VEL
LIN {X 0,Y 457.103,Z 305.805,A -85,B 0,C 180,E1 21005.54,E2 21005.54} C_VEL
LIN {X 0,Y 463.769,Z 323.915,A -85,B 0,C 180,E1 21002.659,E2 21002.659} C_VEL
LIN {X 0,Y 469.458,Z 340.836,A -85,B 0,C 180,E1 21000.272,E2 21000.272} C_VEL
LIN {X 0,Y 473.675,Z 360.592,A -85,B 0,C 180,E1 20999.595,E2 20999.595} C_VEL
LIN {X 0,Y 472.928,Z 415.659,A -85,B 0,C 180,E1 20998.756,E2 20998.756} C_VEL
LIN {X 0,Y 471.972,Z 423.356,A -85,B 0,C 180,E1 20998.706,E2 20998.706} C_VEL
LIN {X 0,Y 466.393,Z 443.845,A -85,B 0,C 180,E1 20998.803,E2 20998.803} C_VEL
LIN {X 0,Y 465.674,Z 450.451,A -85,B 0,C 180,E1 20998.752,E2 20998.752} C_VEL
LIN {X 0,Y 464.448,Z 555.437,A -85,B 0,C 180,E1 20997.136,E2 20997.136} C_VEL
LIN {X 0,Y 463.939,Z 574.591,A -85,B 0,C 180,E1 20996.601,E2 20996.601} C_VEL
LIN {X 0,Y 463.055,Z 592.759,A -85,B 0,C 180,E1 20995.859,E2 20995.859} C_VEL
LIN {X 0,Y 461.864,Z 610.346,A -85,B 0,C 180,E1 20994.896,E2 20994.896} C_VEL
LIN {X 0,Y 460.428,Z 626.775,A -85,B 0,C 180,E1 20993.754,E2 20993.754} C_VEL
LIN {X 0,Y 458.829,Z 642.304,A -85,B 0,C 180,E1 20992.417,E2 20992.417} C_VEL
LIN {X 0,Y 457.058,Z 657.387,A -85,B 0,C 180,E1 20990.823,E2 20990.823} C_VEL
LIN {X 0,Y 455.37,Z 670.816,A -85,B 0,C 180,E1 20989.096,E2 20989.096} C_VEL
LIN {X 0,Y 453.728,Z 683.14,A -85,B 0,C 180,E1 20987.174,E2 20987.174} C_VEL
LIN {X 0,Y 452.311,Z 693.94,A -85,B 0,C 180,E1 20985.12,E2 20985.12} C_VEL
LIN {X 0,Y 451.104,Z 703.269,A -85,B 0,C 180,E1 20982.936,E2 20982.936} C_VEL
LIN {X 0,Y 450.168,Z 711.111,A -85,B 0,C 180,E1 20980.623,E2 20980.623} C_VEL
LIN {X 0,Y 449.509,Z 717.445,A -85,B 0,C 180,E1 20978.176,E2 20978.176} C_VEL
LIN {X 0,Y 449.079,Z 721.959,A -85,B 0,C 180,E1 20975.75,E2 20975.75} C_VEL
LIN {X 0,Y 448.842,Z 724.845,A -85,B 0,C 180,E1 20973.32,E2 20973.32} C_VEL
LIN {X 0,Y 448.752,Z 726.203,A -85,B 0,C 180,E1 20970.766,E2 20970.766} C_VEL
LIN {X 0,Y 448.772,Z 725.9,A -85,B 0,C 180,E1 20968.213,E2 20968.213} C_VEL
LIN {X 0,Y 448.915,Z 723.921,A -85,B 0,C 180,E1 20965.657,E2 20965.657} C_VEL
LIN {X 0,Y 449.237,Z 720.186,A -85,B 0,C 180,E1 20963.097,E2 20963.097} C_VEL
LIN {X 0,Y 449.766,Z 714.892,A -85,B 0,C 180,E1 20960.661,E2 20960.661} C_VEL
LIN {X 0,Y 450.51,Z 708.15,A -85,B 0,C 180,E1 20958.348,E2 20958.348} C_VEL
LIN {X 0,Y 451.518,Z 700.026,A -85,B 0,C 180,E1 20956.164,E2 20956.164} C_VEL
LIN {X 0,Y 452.828,Z 689.922,A -85,B 0,C 180,E1 20953.979,E2 20953.979} C_VEL
LIN {X 0,Y 454.274,Z 679.021,A -85,B 0,C 180,E1 20952.053,E2 20952.053} C_VEL
LIN {X 0,Y 455.974,Z 666.102,A -85,B 0,C 180,E1 20950.172,E2 20950.172} C_VEL
LIN {X 0,Y 457.635,Z 652.624,A -85,B 0,C 180,E1 20948.552,E2 20948.552} C_VEL
LIN {X 0,Y 459.324,Z 637.67,A -85,B 0,C 180,E1 20947.068,E2 20947.068} C_VEL
LIN {X 0,Y 460.868,Z 621.935,A -85,B 0,C 180,E1 20945.794,E2 20945.794} C_VEL
LIN {X 0,Y 462.244,Z 605.266,A -85,B 0,C 180,E1 20944.711,E2 20944.711} C_VEL
LIN {X 0,Y 463.346,Z 587.531,A -85,B 0,C 180,E1 20943.815,E2 20943.815} C_VEL
LIN {X 0,Y 464.133,Z 568.86,A -85,B 0,C 180,E1 20943.125,E2 20943.125} C_VEL
LIN {X 0,Y 464.508,Z 549.822,A -85,B 0,C 180,E1 20942.664,E2 20942.664} C_VEL
LIN {X 0,Y 466.839,Z 360.55,A -85,B 0,C 180,E1 20939.758,E2 20939.758} C_VEL
LIN {X 0,Y 463.216,Z 344.477,A -85,B 0,C 180,E1 20939.185,E2 20939.185} C_VEL
LIN {X 0,Y 461.228,Z 340.497,A -85,B 0,C 180,E1 20938.903,E2 20938.903} C_VEL
LIN {X 0,Y 454.943,Z 322.197,A -85,B 0,C 180,E1 20936.177,E2 20936.177} C_VEL
LIN {X 0,Y 449.159,Z 306.761,A -85,B 0,C 180,E1 20933.614,E2 20933.614} C_VEL
LIN {X 0,Y 449.139,Z 306.517,A -85,B 0,C 180,E1 20930.125,E2 20930.125} C_VEL
LIN {X 0,Y 449.113,Z 306.501,A -85,B 0,C 180,E1 20926.534,E2 20926.534} C_VEL
LIN {X 0,Y 449.102,Z 306.543,A -85,B 0,C 180,E1 20922.908,E2 20922.908} C_VEL
LIN {X 0,Y 449.105,Z 306.541,A -85,B 0,C 180,E1 20919.218,E2 20919.218} C_VEL
LIN {X 0,Y 449.122,Z 306.541,A -85,B 0,C 180,E1 20915.525,E2 20915.525} C_VEL
LIN {X 0,Y 449.14,Z 306.54,A -85,B 0,C 180,E1 20911.748,E2 20911.748} C_VEL
LIN {X 0,Y 449.128,Z 306.534,A -85,B 0,C 180,E1 20908.017,E2 20908.017} C_VEL
LIN {X 0,Y 449.095,Z 306.526,A -85,B 0,C 180,E1 20904.323,E2 20904.323} C_VEL
LIN {X 0,Y 449.08,Z 306.536,A -85,B 0,C 180,E1 20900.733,E2 20900.733} C_VEL
LIN {X 0,Y 449.088,Z 306.544,A -85,B 0,C 180,E1 20897.091,E2 20897.091} C_VEL
LIN {X 0,Y 449.12,Z 306.525,A -85,B 0,C 180,E1 20893.519,E2 20893.519} C_VEL
LIN {X 0,Y 449.112,Z 306.53,A -85,B 0,C 180,E1 20889.742,E2 20889.742} C_VEL
LIN {X 0,Y 449.07,Z 306.544,A -85,B 0,C 180,E1 20886.264,E2 20886.264} C_VEL
LIN {X 0,Y 449.057,Z 306.529,A -85,B 0,C 180,E1 20882.553,E2 20882.553} C_VEL
LIN {X 0,Y 449.072,Z 306.539,A -85,B 0,C 180,E1 20878.98,E2 20878.98} C_VEL
LIN {X 0,Y 449.104,Z 306.54,A -85,B 0,C 180,E1 20875.275,E2 20875.275} C_VEL
LIN {X 0,Y 449.099,Z 306.526,A -85,B 0,C 180,E1 20871.68,E2 20871.68} C_VEL
LIN {X 0,Y 449.077,Z 306.544,A -85,B 0,C 180,E1 20868.05,E2 20868.05} C_VEL
LIN {X 0,Y 449.074,Z 306.544,A -85,B 0,C 180,E1 20864.371,E2 20864.371} C_VEL
LIN {X 0,Y 449.09,Z 306.536,A -85,B 0,C 180,E1 20860.729,E2 20860.729} C_VEL
LIN {X 0,Y 449.126,Z 306.527,A -85,B 0,C 180,E1 20857.071,E2 20857.071} C_VEL
LIN {X 0,Y 449.124,Z 306.531,A -85,B 0,C 180,E1 20853.419,E2 20853.419} C_VEL
LIN {X 0,Y 449.094,Z 306.541,A -85,B 0,C 180,E1 20849.938,E2 20849.938} C_VEL
LIN {X 0,Y 449.093,Z 306.536,A -85,B 0,C 180,E1 20846.179,E2 20846.179} C_VEL
LIN {X 0,Y 449.098,Z 306.518,A -85,B 0,C 180,E1 20842.409,E2 20842.409} C_VEL
LIN {X 0,Y 449.129,Z 306.502,A -85,B 0,C 180,E1 20838.802,E2 20838.802} C_VEL
LIN {X 0,Y 449.137,Z 306.52,A -85,B 0,C 180,E1 20835.065,E2 20835.065} C_VEL
LIN {X 0,Y 449.164,Z 306.836,A -85,B 0,C 180,E1 20834.547,E2 20834.547} C_VEL
LIN {X 0,Y 450.611,Z 310.296,A -85,B 0,C 180,E1 20834.035,E2 20834.035} C_VEL
LIN {X 0,Y 459.097,Z 329.386,A -85,B 0,C 180,E1 20831.574,E2 20831.574} C_VEL
LIN {X 0,Y 467.271,Z 349.616,A -85,B 0,C 180,E1 20829.231,E2 20829.231} C_VEL
LIN {X 0,Y 467.455,Z 351.849,A -85,B 0,C 180,E1 20829.043,E2 20829.043} C_VEL
LIN {X 0,Y 465.163,Z 385.883,A -85,B 0,C 180,E1 20826.644,E2 20826.644} C_VEL
LIN {X 0,Y 468.361,Z 414.894,A -85,B 0,C 180,E1 20825.843,E2 20825.843} C_VEL
LIN {X 0,Y 463.596,Z 639.784,A -85,B 0,C 180,E1 20821.953,E2 20821.953} C_VEL
LIN {X 0,Y 462.571,Z 661.56,A -85,B 0,C 180,E1 20821.407,E2 20821.407} C_VEL
LIN {X 0,Y 461.202,Z 682.982,A -85,B 0,C 180,E1 20820.627,E2 20820.627} C_VEL
LIN {X 0,Y 459.699,Z 703.09,A -85,B 0,C 180,E1 20819.657,E2 20819.657} C_VEL
LIN {X 0,Y 458.115,Z 722.498,A -85,B 0,C 180,E1 20818.481,E2 20818.481} C_VEL
LIN {X 0,Y 456.462,Z 741.224,A -85,B 0,C 180,E1 20817.104,E2 20817.104} C_VEL
LIN {X 0,Y 454.747,Z 760.543,A -85,B 0,C 180,E1 20815.387,E2 20815.387} C_VEL
LIN {X 0,Y 453.188,Z 778.072,A -85,B 0,C 180,E1 20813.536,E2 20813.536} C_VEL
LIN {X 0,Y 451.78,Z 794.389,A -85,B 0,C 180,E1 20811.485,E2 20811.485} C_VEL
LIN {X 0,Y 450.61,Z 808.971,A -85,B 0,C 180,E1 20809.306,E2 20809.306} C_VEL
LIN {X 0,Y 449.729,Z 820.861,A -85,B 0,C 180,E1 20807.198,E2 20807.198} C_VEL
LIN {X 0,Y 449.033,Z 832.082,A -85,B 0,C 180,E1 20804.837,E2 20804.837} C_VEL
LIN {X 0,Y 448.55,Z 841.271,A -85,B 0,C 180,E1 20802.487,E2 20802.487} C_VEL
LIN {X 0,Y 448.267,Z 849.018,A -85,B 0,C 180,E1 20800.019,E2 20800.019} C_VEL
LIN {X 0,Y 448.128,Z 854.858,A -85,B 0,C 180,E1 20797.564,E2 20797.564} C_VEL
LIN {X 0,Y 448.085,Z 859.007,A -85,B 0,C 180,E1 20795.121,E2 20795.121} C_VEL
LIN {X 0,Y 448.079,Z 861.577,A -85,B 0,C 180,E1 20792.686,E2 20792.686} C_VEL
LIN {X 0,Y 448.08,Z 862.524,A -85,B 0,C 180,E1 20790.256,E2 20790.256} C_VEL
LIN {X 0,Y 448.076,Z 861.878,A -85,B 0,C 180,E1 20787.826,E2 20787.826} C_VEL
LIN {X 0,Y 448.072,Z 859.704,A -85,B 0,C 180,E1 20785.392,E2 20785.392} C_VEL
LIN {X 0,Y 448.118,Z 855.896,A -85,B 0,C 180,E1 20782.951,E2 20782.951} C_VEL
LIN {X 0,Y 448.246,Z 850.357,A -85,B 0,C 180,E1 20780.499,E2 20780.499} C_VEL
LIN {X 0,Y 448.482,Z 843.042,A -85,B 0,C 180,E1 20778.034,E2 20778.034} C_VEL
LIN {X 0,Y 448.908,Z 834.248,A -85,B 0,C 180,E1 20775.668,E2 20775.668} C_VEL
LIN {X 0,Y 449.544,Z 823.619,A -85,B 0,C 180,E1 20773.327,E2 20773.327} C_VEL
LIN {X 0,Y 450.454,Z 810.898,A -85,B 0,C 180,E1 20771.01,E2 20771.01} C_VEL
LIN {X 0,Y 451.572,Z 796.731,A -85,B 0,C 180,E1 20768.845,E2 20768.845} C_VEL
LIN {X 0,Y 452.889,Z 781.387,A -85,B 0,C 180,E1 20766.861,E2 20766.861} C_VEL
LIN {X 0,Y 454.387,Z 764.479,A -85,B 0,C 180,E1 20765.009,E2 20765.009} C_VEL
LIN {X 0,Y 456.049,Z 745.912,A -85,B 0,C 180,E1 20763.292,E2 20763.292} C_VEL
LIN {X 0,Y 457.692,Z 727.212,A -85,B 0,C 180,E1 20761.845,E2 20761.845} C_VEL
LIN {X 0,Y 459.337,Z 707.762,A -85,B 0,C 180,E1 20760.604,E2 20760.604} C_VEL
LIN {X 0,Y 460.87,Z 687.741,A -85,B 0,C 180,E1 20759.576,E2 20759.576} C_VEL
LIN {X 0,Y 462.289,Z 666.752,A -85,B 0,C 180,E1 20758.753,E2 20758.753} C_VEL
LIN {X 0,Y 463.451,Z 644.624,A -85,B 0,C 180,E1 20758.143,E2 20758.143} C_VEL
LIN {X 0,Y 468.168,Z 423.727,A -85,B 0,C 180,E1 20754.308,E2 20754.308} C_VEL
LIN {X 0,Y 468.187,Z 411.752,A -85,B 0,C 180,E1 20754.086,E2 20754.086} C_VEL
LIN {X 0,Y 465.121,Z 384.724,A -85,B 0,C 180,E1 20753.302,E2 20753.302} C_VEL
LIN {X 0,Y 467.47,Z 350.191,A -85,B 0,C 180,E1 20750.836,E2 20750.836} C_VEL
LIN {X 0,Y 459.285,Z 329.892,A -85,B 0,C 180,E1 20748.493,E2 20748.493} C_VEL
LIN {X 0,Y 451.764,Z 313.011,A -85,B 0,C 180,E1 20746.33,E2 20746.33} C_VEL
LIN {X 0,Y 449.172,Z 306.891,A -85,B 0,C 180,E1 20745.479,E2 20745.479} C_VEL
LIN {X 0,Y 449.136,Z 306.521,A -85,B 0,C 180,E1 20744.886,E2 20744.886} C_VEL
LIN {X 0,Y 449.13,Z 306.502,A -85,B 0,C 180,E1 20741.198,E2 20741.198} C_VEL
LIN {X 0,Y 449.1,Z 306.518,A -85,B 0,C 180,E1 20737.574,E2 20737.574} C_VEL
LIN {X 0,Y 449.093,Z 306.537,A -85,B 0,C 180,E1 20733.821,E2 20733.821} C_VEL
LIN {X 0,Y 449.096,Z 306.542,A -85,B 0,C 180,E1 20730.062,E2 20730.062} C_VEL
LIN {X 0,Y 449.121,Z 306.533,A -85,B 0,C 180,E1 20726.501,E2 20726.501} C_VEL
LIN {X 0,Y 449.138,Z 306.526,A -85,B 0,C 180,E1 20722.79,E2 20722.79} C_VEL
LIN {X 0,Y 449.102,Z 306.533,A -85,B 0,C 180,E1 20719.103,E2 20719.103} C_VEL
LIN {X 0,Y 449.077,Z 306.543,A -85,B 0,C 180,E1 20715.496,E2 20715.496} C_VEL
LIN {X 0,Y 449.072,Z 306.543,A -85,B 0,C 180,E1 20711.689,E2 20711.689} C_VEL
LIN {X 0,Y 449.083,Z 306.529,A -85,B 0,C 180,E1 20708.063,E2 20708.063} C_VEL
LIN {X 0,Y 449.113,Z 306.537,A -85,B 0,C 180,E1 20704.469,E2 20704.469} C_VEL
LIN {X 0,Y 449.111,Z 306.539,A -85,B 0,C 180,E1 20700.638,E2 20700.638} C_VEL
LIN {X 0,Y 449.073,Z 306.527,A -85,B 0,C 180,E1 20696.937,E2 20696.937} C_VEL
LIN {X 0,Y 449.06,Z 306.544,A -85,B 0,C 180,E1 20693.351,E2 20693.351} C_VEL
LIN {X 0,Y 449.067,Z 306.543,A -85,B 0,C 180,E1 20689.61,E2 20689.61} C_VEL
LIN {X 0,Y 449.091,Z 306.525,A -85,B 0,C 180,E1 20685.955,E2 20685.955} C_VEL
LIN {X 0,Y 449.124,Z 306.538,A -85,B 0,C 180,E1 20682.327,E2 20682.327} C_VEL
LIN {X 0,Y 449.106,Z 306.537,A -85,B 0,C 180,E1 20678.585,E2 20678.585} C_VEL
LIN {X 0,Y 449.081,Z 306.527,A -85,B 0,C 180,E1 20674.974,E2 20674.974} C_VEL
LIN {X 0,Y 449.083,Z 306.537,A -85,B 0,C 180,E1 20671.255,E2 20671.255} C_VEL
LIN {X 0,Y 449.108,Z 306.54,A -85,B 0,C 180,E1 20667.702,E2 20667.702} C_VEL
LIN {X 0,Y 449.135,Z 306.541,A -85,B 0,C 180,E1 20664.005,E2 20664.005} C_VEL
LIN {X 0,Y 449.131,Z 306.544,A -85,B 0,C 180,E1 20660.288,E2 20660.288} C_VEL
LIN {X 0,Y 449.102,Z 306.545,A -85,B 0,C 180,E1 20656.708,E2 20656.708} C_VEL
LIN {X 0,Y 449.097,Z 306.508,A -85,B 0,C 180,E1 20652.942,E2 20652.942} C_VEL
LIN {X 0,Y 449.106,Z 306.512,A -85,B 0,C 180,E1 20649.216,E2 20649.216} C_VEL
LIN {X 0,Y 449.165,Z 306.808,A -85,B 0,C 180,E1 20646.266,E2 20646.266} C_VEL
LIN {X 0,Y 455.602,Z 324.164,A -85,B 0,C 180,E1 20643.424,E2 20643.424} C_VEL
LIN {X 0,Y 461.389,Z 340.979,A -85,B 0,C 180,E1 20640.949,E2 20640.949} C_VEL
LIN {X 0,Y 463.678,Z 345.93,A -85,B 0,C 180,E1 20640.654,E2 20640.654} C_VEL
LIN {X 0,Y 466.947,Z 362.206,A -85,B 0,C 180,E1 20640.105,E2 20640.105} C_VEL
LIN {X 0,Y 465.674,Z 450.451,A -85,B 0,C 180,E1 20638.752,E2 20638.752} C_VEL
LIN {X 0,Y 464.731,Z 458.149,A -85,B 0,C 180,E1 20638.701,E2 20638.701} C_VEL
LIN {X 0,Y 459.143,Z 478.637,A -85,B 0,C 180,E1 20638.803,E2 20638.803} C_VEL
LIN {X 0,Y 458.427,Z 485.244,A -85,B 0,C 180,E1 20638.751,E2 20638.751} C_VEL
LIN {X 0,Y 457.554,Z 556.603,A -85,B 0,C 180,E1 20637.624,E2 20637.624} C_VEL
LIN {X 0,Y 457.008,Z 575.637,A -85,B 0,C 180,E1 20637.082,E2 20637.082} C_VEL
LIN {X 0,Y 456.071,Z 593.857,A -85,B 0,C 180,E1 20636.326,E2 20636.326} C_VEL
LIN {X 0,Y 454.859,Z 610.95,A -85,B 0,C 180,E1 20635.381,E2 20635.381} C_VEL
LIN {X 0,Y 453.336,Z 627.514,A -85,B 0,C 180,E1 20634.219,E2 20634.219} C_VEL
LIN {X 0,Y 451.566,Z 643.756,A -85,B 0,C 180,E1 20632.797,E2 20632.797} C_VEL
LIN {X 0,Y 449.774,Z 658.25,A -85,B 0,C 180,E1 20631.244,E2 20631.244} C_VEL
LIN {X 0,Y 447.917,Z 672.162,A -85,B 0,C 180,E1 20629.426,E2 20629.426} C_VEL
LIN {X 0,Y 446.18,Z 684.452,A -85,B 0,C 180,E1 20627.474,E2 20627.474} C_VEL
LIN {X 0,Y 444.671,Z 695.225,A -85,B 0,C 180,E1 20625.386,E2 20625.386} C_VEL
LIN {X 0,Y 443.385,Z 704.531,A -85,B 0,C 180,E1 20623.165,E2 20623.165} C_VEL
LIN {X 0,Y 442.379,Z 712.355,A -85,B 0,C 180,E1 20620.812,E2 20620.812} C_VEL
LIN {X 0,Y 441.688,Z 718.493,A -85,B 0,C 180,E1 20618.408,E2 20618.408} C_VEL
LIN {X 0,Y 441.222,Z 722.989,A -85,B 0,C 180,E1 20615.983,E2 20615.983} C_VEL
LIN {X 0,Y 440.953,Z 725.95,A -85,B 0,C 180,E1 20613.51,E2 20613.51} C_VEL
LIN {X 0,Y 440.844,Z 727.386,A -85,B 0,C 180,E1 20610.91,E2 20610.91} C_VEL
LIN {X 0,Y 440.863,Z 727.163,A -85,B 0,C 180,E1 20608.311,E2 20608.311} C_VEL
LIN {X 0,Y 441.011,Z 725.273,A -85,B 0,C 180,E1 20605.709,E2 20605.709} C_VEL
LIN {X 0,Y 441.351,Z 721.635,A -85,B 0,C 180,E1 20603.104,E2 20603.104} C_VEL
LIN {X 0,Y 441.945,Z 716.126,A -85,B 0,C 180,E1 20600.494,E2 20600.494} C_VEL
LIN {X 0,Y 442.749,Z 709.4,A -85,B 0,C 180,E1 20598.141,E2 20598.141} C_VEL
LIN {X 0,Y 443.829,Z 701.296,A -85,B 0,C 180,E1 20595.919,E2 20595.919} C_VEL
LIN {X 0,Y 445.225,Z 691.214,A -85,B 0,C 180,E1 20593.697,E2 20593.697} C_VEL
LIN {X 0,Y 446.762,Z 680.343,A -85,B 0,C 180,E1 20591.741,E2 20591.741} C_VEL
LIN {X 0,Y 448.47,Z 668.121,A -85,B 0,C 180,E1 20589.92,E2 20589.92} C_VEL
LIN {X 0,Y 450.259,Z 654.459,A -85,B 0,C 180,E1 20588.233,E2 20588.233} C_VEL
LIN {X 0,Y 452.093,Z 639.146,A -85,B 0,C 180,E1 20586.68,E2 20586.68} C_VEL
LIN {X 0,Y 453.805,Z 622.633,A -85,B 0,C 180,E1 20585.323,E2 20585.323} C_VEL
LIN {X 0,Y 455.262,Z 605.77,A -85,B 0,C 180,E1 20584.218,E2 20584.218} C_VEL
LIN {X 0,Y 456.418,Z 588.013,A -85,B 0,C 180,E1 20583.316,E2 20583.316} C_VEL
LIN {X 0,Y 457.233,Z 569.486,A -85,B 0,C 180,E1 20582.627,E2 20582.627} C_VEL
LIN {X 0,Y 457.625,Z 550.546,A -85,B 0,C 180,E1 20582.164,E2 20582.164} C_VEL
LIN {X 0,Y 460.162,Z 362.043,A -85,B 0,C 180,E1 20579.23,E2 20579.23} C_VEL
LIN {X 0,Y 457.006,Z 348.141,A -85,B 0,C 180,E1 20578.719,E2 20578.719} C_VEL
LIN {X 0,Y 453.359,Z 341.115,A -85,B 0,C 180,E1 20578.234,E2 20578.234} C_VEL
LIN {X 0,Y 447.108,Z 323.226,A -85,B 0,C 180,E1 20575.495,E2 20575.495} C_VEL
LIN {X 0,Y 442.158,Z 310.486,A -85,B 0,C 180,E1 20573.347,E2 20573.347} C_VEL
LIN {X 0,Y 441.194,Z 307.667,A -85,B 0,C 180,E1 20572.811,E2 20572.811} C_VEL
LIN {X 0,Y 441.17,Z 307.534,A -85,B 0,C 180,E1 20569.083,E2 20569.083} C_VEL
LIN {X 0,Y 441.171,Z 307.493,A -85,B 0,C 180,E1 20565.368,E2 20565.368} C_VEL
LIN {X 0,Y 441.191,Z 307.519,A -85,B 0,C 180,E1 20561.596,E2 20561.596} C_VEL
LIN {X 0,Y 441.202,Z 307.516,A -85,B 0,C 180,E1 20557.89,E2 20557.89} C_VEL
LIN {X 0,Y 441.181,Z 307.518,A -85,B 0,C 180,E1 20554.189,E2 20554.189} C_VEL
LIN {X 0,Y 441.156,Z 307.527,A -85,B 0,C 180,E1 20550.51,E2 20550.51} C_VEL
LIN {X 0,Y 441.148,Z 307.532,A -85,B 0,C 180,E1 20546.81,E2 20546.81} C_VEL
LIN {X 0,Y 441.151,Z 307.533,A -85,B 0,C 180,E1 20543.05,E2 20543.05} C_VEL
LIN {X 0,Y 441.175,Z 307.513,A -85,B 0,C 180,E1 20539.461,E2 20539.461} C_VEL
LIN {X 0,Y 441.184,Z 307.523,A -85,B 0,C 180,E1 20535.781,E2 20535.781} C_VEL
LIN {X 0,Y 441.144,Z 307.529,A -85,B 0,C 180,E1 20532.169,E2 20532.169} C_VEL
LIN {X 0,Y 441.126,Z 307.513,A -85,B 0,C 180,E1 20528.472,E2 20528.472} C_VEL
LIN {X 0,Y 441.123,Z 307.531,A -85,B 0,C 180,E1 20524.681,E2 20524.681} C_VEL
LIN {X 0,Y 441.137,Z 307.533,A -85,B 0,C 180,E1 20521.039,E2 20521.039} C_VEL
LIN {X 0,Y 441.166,Z 307.512,A -85,B 0,C 180,E1 20517.402,E2 20517.402} C_VEL
LIN {X 0,Y 441.167,Z 307.528,A -85,B 0,C 180,E1 20513.624,E2 20513.624} C_VEL
LIN {X 0,Y 441.141,Z 307.529,A -85,B 0,C 180,E1 20509.949,E2 20509.949} C_VEL
LIN {X 0,Y 441.132,Z 307.515,A -85,B 0,C 180,E1 20506.232,E2 20506.232} C_VEL
LIN {X 0,Y 441.136,Z 307.526,A -85,B 0,C 180,E1 20502.455,E2 20502.455} C_VEL
LIN {X 0,Y 441.155,Z 307.53,A -85,B 0,C 180,E1 20498.738,E2 20498.738} C_VEL
LIN {X 0,Y 441.188,Z 307.531,A -85,B 0,C 180,E1 20495.069,E2 20495.069} C_VEL
LIN {X 0,Y 441.203,Z 307.527,A -85,B 0,C 180,E1 20491.282,E2 20491.282} C_VEL
LIN {X 0,Y 441.177,Z 307.53,A -85,B 0,C 180,E1 20487.512,E2 20487.512} C_VEL
LIN {X 0,Y 441.158,Z 307.485,A -85,B 0,C 180,E1 20483.787,E2 20483.787} C_VEL
LIN {X 0,Y 441.158,Z 307.518,A -85,B 0,C 180,E1 20480.104,E2 20480.104} C_VEL
LIN {X 0,Y 441.172,Z 307.517,A -85,B 0,C 180,E1 20476.451,E2 20476.451} C_VEL
LIN {X 0,Y 441.225,Z 307.774,A -85,B 0,C 180,E1 20475.36,E2 20475.36} C_VEL
LIN {X 0,Y 442.653,Z 311.217,A -85,B 0,C 180,E1 20474.826,E2 20474.826} C_VEL
LIN {X 0,Y 451.265,Z 330.255,A -85,B 0,C 180,E1 20472.266,E2 20472.266} C_VEL
LIN {X 0,Y 459.55,Z 350.659,A -85,B 0,C 180,E1 20469.823,E2 20469.823} C_VEL
LIN {X 0,Y 460.574,Z 353.601,A -85,B 0,C 180,E1 20469.498,E2 20469.498} C_VEL
LIN {X 0,Y 458.278,Z 385.51,A -85,B 0,C 180,E1 20467.218,E2 20467.218} C_VEL
LIN {X 0,Y 461.594,Z 416.023,A -85,B 0,C 180,E1 20466.357,E2 20466.357} C_VEL
LIN {X 0,Y 456.582,Z 638.411,A -85,B 0,C 180,E1 20462.453,E2 20462.453} C_VEL
LIN {X 0,Y 455.51,Z 660.4,A -85,B 0,C 180,E1 20461.896,E2 20461.896} C_VEL
LIN {X 0,Y 454.066,Z 681.451,A -85,B 0,C 180,E1 20461.125,E2 20461.125} C_VEL
LIN {X 0,Y 452.521,Z 701.039,A -85,B 0,C 180,E1 20460.176,E2 20460.176} C_VEL
LIN {X 0,Y 450.788,Z 720.778,A -85,B 0,C 180,E1 20458.972,E2 20458.972} C_VEL
LIN {X 0,Y 448.957,Z 740.152,A -85,B 0,C 180,E1 20457.523,E2 20457.523} C_VEL
LIN {X 0,Y 447.195,Z 758.68,A -85,B 0,C 180,E1 20455.847,E2 20455.847} C_VEL
LIN {X 0,Y 445.465,Z 776.639,A -85,B 0,C 180,E1 20453.91,E2 20453.91} C_VEL
LIN {X 0,Y 443.924,Z 793.523,A -85,B 0,C 180,E1 20451.746,E2 20451.746} C_VEL
LIN {X 0,Y 442.7,Z 808.087,A -85,B 0,C 180,E1 20449.527,E2 20449.527} C_VEL
LIN {X 0,Y 441.739,Z 820.649,A -85,B 0,C 180,E1 20447.248,E2 20447.248} C_VEL
LIN {X 0,Y 441.072,Z 831.137,A -85,B 0,C 180,E1 20444.976,E2 20444.976} C_VEL
LIN {X 0,Y 440.59,Z 840.306,A -85,B 0,C 180,E1 20442.583,E2 20442.583} C_VEL
LIN {X 0,Y 440.322,Z 847.692,A -85,B 0,C 180,E1 20440.202,E2 20440.202} C_VEL
LIN {X 0,Y 440.193,Z 853.586,A -85,B 0,C 180,E1 20437.701,E2 20437.701} C_VEL
LIN {X 0,Y 440.159,Z 857.778,A -85,B 0,C 180,E1 20435.213,E2 20435.213} C_VEL
LIN {X 0,Y 440.166,Z 860.368,A -85,B 0,C 180,E1 20432.734,E2 20432.734} C_VEL
LIN {X 0,Y 440.17,Z 861.323,A -85,B 0,C 180,E1 20430.26,E2 20430.26} C_VEL
LIN {X 0,Y 440.163,Z 860.669,A -85,B 0,C 180,E1 20427.787,E2 20427.787} C_VEL
LIN {X 0,Y 440.152,Z 858.475,A -85,B 0,C 180,E1 20425.309,E2 20425.309} C_VEL
LIN {X 0,Y 440.18,Z 854.64,A -85,B 0,C 180,E1 20422.823,E2 20422.823} C_VEL
LIN {X 0,Y 440.299,Z 849.047,A -85,B 0,C 180,E1 20420.326,E2 20420.326} C_VEL
LIN {X 0,Y 440.536,Z 841.653,A -85,B 0,C 180,E1 20417.815,E2 20417.815} C_VEL
LIN {X 0,Y 440.979,Z 832.844,A -85,B 0,C 180,E1 20415.424,E2 20415.424} C_VEL
LIN {X 0,Y 441.647,Z 822.041,A -85,B 0,C 180,E1 20413.02,E2 20413.02} C_VEL
LIN {X 0,Y 442.571,Z 809.682,A -85,B 0,C 180,E1 20410.741,E2 20410.741} C_VEL
LIN {X 0,Y 443.709,Z 795.842,A -85,B 0,C 180,E1 20408.59,E2 20408.59} C_VEL
LIN {X 0,Y 445.087,Z 780.574,A -85,B 0,C 180,E1 20406.571,E2 20406.571} C_VEL
LIN {X 0,Y 446.736,Z 763.246,A -85,B 0,C 180,E1 20404.622,E2 20404.622} C_VEL
LIN {X 0,Y 448.509,Z 744.809,A -85,B 0,C 180,E1 20402.879,E2 20402.879} C_VEL
LIN {X 0,Y 450.297,Z 726.014,A -85,B 0,C 180,E1 20401.398,E2 20401.398} C_VEL
LIN {X 0,Y 452.02,Z 706.85,A -85,B 0,C 180,E1 20400.153,E2 20400.153} C_VEL
LIN {X 0,Y 453.682,Z 686.699,A -85,B 0,C 180,E1 20399.104,E2 20399.104} C_VEL
LIN {X 0,Y 455.181,Z 665.713,A -85,B 0,C 180,E1 20398.269,E2 20398.269} C_VEL
LIN {X 0,Y 456.417,Z 643.585,A -85,B 0,C 180,E1 20397.652,E2 20397.652} C_VEL
LIN {X 0,Y 461.361,Z 425.998,A -85,B 0,C 180,E1 20393.816,E2 20393.816} C_VEL
LIN {X 0,Y 461.425,Z 412.906,A -85,B 0,C 180,E1 20393.572,E2 20393.572} C_VEL
LIN {X 0,Y 458.225,Z 384.258,A -85,B 0,C 180,E1 20392.727,E2 20392.727} C_VEL
LIN {X 0,Y 460.497,Z 353.204,A -85,B 0,C 180,E1 20390.469,E2 20390.469} C_VEL
LIN {X 0,Y 452.108,Z 332.26,A -85,B 0,C 180,E1 20387.994,E2 20387.994} C_VEL
LIN {X 0,Y 444.308,Z 314.885,A -85,B 0,C 180,E1 20385.694,E2 20385.694} C_VEL
LIN {X 0,Y 441.262,Z 307.966,A -85,B 0,C 180,E1 20384.704,E2 20384.704} C_VEL
LIN {X 0,Y 441.179,Z 307.533,A -85,B 0,C 180,E1 20384.449,E2 20384.449} C_VEL
LIN {X 0,Y 441.197,Z 307.494,A -85,B 0,C 180,E1 20380.743,E2 20380.743} C_VEL
LIN {X 0,Y 441.19,Z 307.49,A -85,B 0,C 180,E1 20377.072,E2 20377.072} C_VEL
LIN {X 0,Y 441.167,Z 307.529,A -85,B 0,C 180,E1 20373.417,E2 20373.417} C_VEL
LIN {X 0,Y 441.151,Z 307.533,A -85,B 0,C 180,E1 20369.759,E2 20369.759} C_VEL
LIN {X 0,Y 441.155,Z 307.531,A -85,B 0,C 180,E1 20366.084,E2 20366.084} C_VEL
LIN {X 0,Y 441.172,Z 307.521,A -85,B 0,C 180,E1 20362.38,E2 20362.38} C_VEL
LIN {X 0,Y 441.188,Z 307.515,A -85,B 0,C 180,E1 20358.635,E2 20358.635} C_VEL
LIN {X 0,Y 441.179,Z 307.523,A -85,B 0,C 180,E1 20354.838,E2 20354.838} C_VEL
LIN {X 0,Y 441.149,Z 307.531,A -85,B 0,C 180,E1 20351.107,E2 20351.107} C_VEL
LIN {X 0,Y 441.129,Z 307.523,A -85,B 0,C 180,E1 20347.423,E2 20347.423} C_VEL
LIN {X 0,Y 441.123,Z 307.523,A -85,B 0,C 180,E1 20343.638,E2 20343.638} C_VEL
LIN {X 0,Y 441.138,Z 307.535,A -85,B 0,C 180,E1 20340,E2 20340} C_VEL
LIN {X 0,Y 441.164,Z 307.515,A -85,B 0,C 180,E1 20336.361,E2 20336.361} C_VEL
LIN {X 0,Y 441.166,Z 307.519,A -85,B 0,C 180,E1 20332.577,E2 20332.577} C_VEL
LIN {X 0,Y 441.141,Z 307.533,A -85,B 0,C 180,E1 20328.892,E2 20328.892} C_VEL
LIN {X 0,Y 441.129,Z 307.517,A -85,B 0,C 180,E1 20325.294,E2 20325.294} C_VEL
LIN {X 0,Y 441.137,Z 307.525,A -85,B 0,C 180,E1 20321.499,E2 20321.499} C_VEL
LIN {X 0,Y 441.166,Z 307.531,A -85,B 0,C 180,E1 20317.9,E2 20317.9} C_VEL
LIN {X 0,Y 441.188,Z 307.518,A -85,B 0,C 180,E1 20314.206,E2 20314.206} C_VEL
LIN {X 0,Y 441.175,Z 307.517,A -85,B 0,C 180,E1 20310.488,E2 20310.488} C_VEL
LIN {X 0,Y 441.151,Z 307.527,A -85,B 0,C 180,E1 20306.892,E2 20306.892} C_VEL
LIN {X 0,Y 441.152,Z 307.532,A -85,B 0,C 180,E1 20303.086,E2 20303.086} C_VEL
LIN {X 0,Y 441.166,Z 307.528,A -85,B 0,C 180,E1 20299.396,E2 20299.396} C_VEL
LIN {X 0,Y 441.189,Z 307.518,A -85,B 0,C 180,E1 20295.732,E2 20295.732} C_VEL
LIN {X 0,Y 441.199,Z 307.512,A -85,B 0,C 180,E1 20291.953,E2 20291.953} C_VEL
LIN {X 0,Y 441.194,Z 307.492,A -85,B 0,C 180,E1 20288.15,E2 20288.15} C_VEL
LIN {X 0,Y 441.209,Z 307.82,A -85,B 0,C 180,E1 20287.029,E2 20287.029} C_VEL
LIN {X 0,Y 447.654,Z 324.815,A -85,B 0,C 180,E1 20284.153,E2 20284.153} C_VEL
LIN {X 0,Y 453.387,Z 341.24,A -85,B 0,C 180,E1 20281.651,E2 20281.651} C_VEL
LIN {X 0,Y 457.468,Z 349.456,A -85,B 0,C 180,E1 20281.119,E2 20281.119} C_VEL
LIN {X 0,Y 460.259,Z 363.748,A -85,B 0,C 180,E1 20280.631,E2 20280.631} C_VEL
LIN {X 0,Y 458.427,Z 485.244,A -85,B 0,C 180,E1 20278.751,E2 20278.751} C_VEL
LIN {X 0,Y 457.493,Z 492.941,A -85,B 0,C 180,E1 20278.699,E2 20278.699} C_VEL
LIN {X 0,Y 451.905,Z 513.429,A -85,B 0,C 180,E1 20278.802,E2 20278.802} C_VEL
LIN {X 0,Y 451.164,Z 520.038,A -85,B 0,C 180,E1 20278.752,E2 20278.752} C_VEL
LIN {X 0,Y 450.675,Z 558.225,A -85,B 0,C 180,E1 20278.114,E2 20278.114} C_VEL
LIN {X 0,Y 450.095,Z 576.922,A -85,B 0,C 180,E1 20277.568,E2 20277.568} C_VEL
LIN {X 0,Y 449.101,Z 595.146,A -85,B 0,C 180,E1 20276.797,E2 20276.797} C_VEL
LIN {X 0,Y 447.783,Z 612.586,A -85,B 0,C 180,E1 20275.811,E2 20275.811} C_VEL
LIN {X 0,Y 446.132,Z 629.477,A -85,B 0,C 180,E1 20274.596,E2 20274.596} C_VEL
LIN {X 0,Y 444.321,Z 645.19,A -85,B 0,C 180,E1 20273.191,E2 20273.191} C_VEL
LIN {X 0,Y 442.435,Z 659.626,A -85,B 0,C 180,E1 20271.614,E2 20271.614} C_VEL
LIN {X 0,Y 440.617,Z 672.62,A -85,B 0,C 180,E1 20269.9,E2 20269.9} C_VEL
LIN {X 0,Y 438.761,Z 685.034,A -85,B 0,C 180,E1 20267.917,E2 20267.917} C_VEL
LIN {X 0,Y 437.134,Z 695.913,A -85,B 0,C 180,E1 20265.794,E2 20265.794} C_VEL
LIN {X 0,Y 435.747,Z 705.314,A -85,B 0,C 180,E1 20263.535,E2 20263.535} C_VEL
LIN {X 0,Y 434.648,Z 713.225,A -85,B 0,C 180,E1 20261.141,E2 20261.141} C_VEL
LIN {X 0,Y 433.863,Z 719.607,A -85,B 0,C 180,E1 20258.615,E2 20258.615} C_VEL
LIN {X 0,Y 433.335,Z 724.297,A -85,B 0,C 180,E1 20256.025,E2 20256.025} C_VEL
LIN {X 0,Y 433.043,Z 727.257,A -85,B 0,C 180,E1 20253.442,E2 20253.442} C_VEL
LIN {X 0,Y 432.935,Z 728.607,A -85,B 0,C 180,E1 20250.794,E2 20250.794} C_VEL
LIN {X 0,Y 432.96,Z 728.305,A -85,B 0,C 180,E1 20248.147,E2 20248.147} C_VEL
LIN {X 0,Y 433.131,Z 726.337,A -85,B 0,C 180,E1 20245.499,E2 20245.499} C_VEL
LIN {X 0,Y 433.513,Z 722.623,A -85,B 0,C 180,E1 20242.846,E2 20242.846} C_VEL
LIN {X 0,Y 434.128,Z 717.343,A -85,B 0,C 180,E1 20240.316,E2 20240.316} C_VEL
LIN {X 0,Y 435.05,Z 710.224,A -85,B 0,C 180,E1 20237.794,E2 20237.794} C_VEL
LIN {X 0,Y 436.226,Z 702.029,A -85,B 0,C 180,E1 20235.533,E2 20235.533} C_VEL
LIN {X 0,Y 437.631,Z 692.499,A -85,B 0,C 180,E1 20233.406,E2 20233.406} C_VEL
LIN {X 0,Y 439.261,Z 681.655,A -85,B 0,C 180,E1 20231.418,E2 20231.418} C_VEL
LIN {X 0,Y 441.063,Z 669.469,A -85,B 0,C 180,E1 20229.568,E2 20229.568} C_VEL
LIN {X 0,Y 443.026,Z 655.276,A -85,B 0,C 180,E1 20227.789,E2 20227.789} C_VEL
LIN {X 0,Y 444.968,Z 639.901,A -85,B 0,C 180,E1 20226.213,E2 20226.213} C_VEL
LIN {X 0,Y 446.682,Z 624.188,A -85,B 0,C 180,E1 20224.902,E2 20224.902} C_VEL
LIN {X 0,Y 448.259,Z 606.922,A -85,B 0,C 180,E1 20223.75,E2 20223.75} C_VEL
LIN {X 0,Y 449.453,Z 589.653,A -85,B 0,C 180,E1 20222.855,E2 20222.855} C_VEL
LIN {X 0,Y 450.342,Z 570.833,A -85,B 0,C 180,E1 20222.138,E2 20222.138} C_VEL
LIN {X 0,Y 450.77,Z 551.683,A -85,B 0,C 180,E1 20221.658,E2 20221.658} C_VEL
LIN {X 0,Y 453.513,Z 363.494,A -85,B 0,C 180,E1 20218.685,E2 20218.685} C_VEL
LIN {X 0,Y 450.831,Z 351.762,A -85,B 0,C 180,E1 20218.24,E2 20218.24} C_VEL
LIN {X 0,Y 445.523,Z 341.845,A -85,B 0,C 180,E1 20217.548,E2 20217.548} C_VEL
LIN {X 0,Y 439.445,Z 324.714,A -85,B 0,C 180,E1 20214.856,E2 20214.856} C_VEL
LIN {X 0,Y 433.917,Z 310.839,A -85,B 0,C 180,E1 20212.436,E2 20212.436} C_VEL
LIN {X 0,Y 433.292,Z 308.724,A -85,B 0,C 180,E1 20212.037,E2 20212.037} C_VEL
LIN {X 0,Y 433.254,Z 308.51,A -85,B 0,C 180,E1 20208.347,E2 20208.347} C_VEL
LIN {X 0,Y 433.238,Z 308.496,A -85,B 0,C 180,E1 20204.511,E2 20204.511} C_VEL
LIN {X 0,Y 433.222,Z 308.514,A -85,B 0,C 180,E1 20200.78,E2 20200.78} C_VEL
LIN {X 0,Y 433.22,Z 308.515,A -85,B 0,C 180,E1 20197.01,E2 20197.01} C_VEL
LIN {X 0,Y 433.228,Z 308.509,A -85,B 0,C 180,E1 20193.318,E2 20193.318} C_VEL
LIN {X 0,Y 433.251,Z 308.503,A -85,B 0,C 180,E1 20189.596,E2 20189.596} C_VEL
LIN {X 0,Y 433.252,Z 308.508,A -85,B 0,C 180,E1 20185.84,E2 20185.84} C_VEL
LIN {X 0,Y 433.231,Z 308.52,A -85,B 0,C 180,E1 20182.098,E2 20182.098} C_VEL
LIN {X 0,Y 433.205,Z 308.513,A -85,B 0,C 180,E1 20178.434,E2 20178.434} C_VEL
LIN {X 0,Y 433.195,Z 308.504,A -85,B 0,C 180,E1 20174.708,E2 20174.708} C_VEL
LIN {X 0,Y 433.198,Z 308.52,A -85,B 0,C 180,E1 20170.91,E2 20170.91} C_VEL
LIN {X 0,Y 433.22,Z 308.51,A -85,B 0,C 180,E1 20167.293,E2 20167.293} C_VEL
LIN {X 0,Y 433.229,Z 308.502,A -85,B 0,C 180,E1 20163.573,E2 20163.573} C_VEL
LIN {X 0,Y 433.204,Z 308.523,A -85,B 0,C 180,E1 20159.868,E2 20159.868} C_VEL
LIN {X 0,Y 433.186,Z 308.511,A -85,B 0,C 180,E1 20156.162,E2 20156.162} C_VEL
LIN {X 0,Y 433.185,Z 308.509,A -85,B 0,C 180,E1 20152.44,E2 20152.44} C_VEL
LIN {X 0,Y 433.199,Z 308.521,A -85,B 0,C 180,E1 20148.686,E2 20148.686} C_VEL
LIN {X 0,Y 433.226,Z 308.516,A -85,B 0,C 180,E1 20145.02,E2 20145.02} C_VEL
LIN {X 0,Y 433.248,Z 308.503,A -85,B 0,C 180,E1 20141.29,E2 20141.29} C_VEL
LIN {X 0,Y 433.243,Z 308.506,A -85,B 0,C 180,E1 20137.474,E2 20137.474} C_VEL
LIN {X 0,Y 433.217,Z 308.517,A -85,B 0,C 180,E1 20133.844,E2 20133.844} C_VEL
LIN {X 0,Y 433.211,Z 308.521,A -85,B 0,C 180,E1 20130.203,E2 20130.203} C_VEL
LIN {X 0,Y 433.219,Z 308.518,A -85,B 0,C 180,E1 20126.424,E2 20126.424} C_VEL
LIN {X 0,Y 433.241,Z 308.48,A -85,B 0,C 180,E1 20122.768,E2 20122.768} C_VEL
LIN {X 0,Y 433.261,Z 308.478,A -85,B 0,C 180,E1 20119.05,E2 20119.05} C_VEL
LIN {X 0,Y 433.246,Z 308.659,A -85,B 0,C 180,E1 20116.247,E2 20116.247} C_VEL
LIN {X 0,Y 433.614,Z 310.179,A -85,B 0,C 180,E1 20115.965,E2 20115.965} C_VEL
LIN {X 0,Y 437.237,Z 317.665,A -85,B 0,C 180,E1 20114.855,E2 20114.855} C_VEL
LIN {X 0,Y 445.378,Z 335.804,A -85,B 0,C 180,E1 20112.389,E2 20112.389} C_VEL
LIN {X 0,Y 453.62,Z 356.435,A -85,B 0,C 180,E1 20109.888,E2 20109.888} C_VEL
LIN {X 0,Y 451.434,Z 385.093,A -85,B 0,C 180,E1 20107.81,E2 20107.81} C_VEL
LIN {X 0,Y 454.868,Z 417.101,A -85,B 0,C 180,E1 20106.888,E2 20106.888} C_VEL
LIN {X 0,Y 449.597,Z 637.589,A -85,B 0,C 180,E1 20102.959,E2 20102.959} C_VEL
LIN {X 0,Y 448.473,Z 659.52,A -85,B 0,C 180,E1 20102.395,E2 20102.395} C_VEL
LIN {X 0,Y 446.911,Z 680.761,A -85,B 0,C 180,E1 20101.605,E2 20101.605} C_VEL
LIN {X 0,Y 445.281,Z 700.245,A -85,B 0,C 180,E1 20100.644,E2 20100.644} C_VEL
LIN {X 0,Y 443.452,Z 719.693,A -85,B 0,C 180,E1 20099.44,E2 20099.44} C_VEL
LIN {X 0,Y 441.492,Z 739.191,A -85,B 0,C 180,E1 20097.955,E2 20097.955} C_VEL
LIN {X 0,Y 439.603,Z 757.767,A -85,B 0,C 180,E1 20096.243,E2 20096.243} C_VEL
LIN {X 0,Y 437.756,Z 775.628,A -85,B 0,C 180,E1 20094.275,E2 20094.275} C_VEL
LIN {X 0,Y 436.179,Z 791.723,A -85,B 0,C 180,E1 20092.167,E2 20092.167} C_VEL
LIN {X 0,Y 434.853,Z 806.474,A -85,B 0,C 180,E1 20089.879,E2 20089.879} C_VEL
LIN {X 0,Y 433.845,Z 819.048,A -85,B 0,C 180,E1 20087.572,E2 20087.572} C_VEL
LIN {X 0,Y 433.139,Z 829.782,A -85,B 0,C 180,E1 20085.224,E2 20085.224} C_VEL
LIN {X 0,Y 432.642,Z 839.047,A -85,B 0,C 180,E1 20082.771,E2 20082.771} C_VEL
LIN {X 0,Y 432.381,Z 846.347,A -85,B 0,C 180,E1 20080.391,E2 20080.391} C_VEL
LIN {X 0,Y 432.255,Z 852.295,A -85,B 0,C 180,E1 20077.844,E2 20077.844} C_VEL
LIN {X 0,Y 432.237,Z 856.537,A -85,B 0,C 180,E1 20075.309,E2 20075.309} C_VEL
LIN {X 0,Y 432.253,Z 859.158,A -85,B 0,C 180,E1 20072.784,E2 20072.784} C_VEL
LIN {X 0,Y 432.26,Z 860.121,A -85,B 0,C 180,E1 20070.265,E2 20070.265} C_VEL
LIN {X 0,Y 432.25,Z 859.462,A -85,B 0,C 180,E1 20067.746,E2 20067.746} C_VEL
LIN {X 0,Y 432.232,Z 857.242,A -85,B 0,C 180,E1 20065.223,E2 20065.223} C_VEL
LIN {X 0,Y 432.24,Z 853.371,A -85,B 0,C 180,E1 20062.691,E2 20062.691} C_VEL
LIN {X 0,Y 432.348,Z 847.66,A -85,B 0,C 180,E1 20060.122,E2 20060.122} C_VEL
LIN {X 0,Y 432.588,Z 840.256,A -85,B 0,C 180,E1 20057.587,E2 20057.587} C_VEL
LIN {X 0,Y 433.08,Z 830.793,A -85,B 0,C 180,E1 20055.015,E2 20055.015} C_VEL
LIN {X 0,Y 433.785,Z 819.943,A -85,B 0,C 180,E1 20052.602,E2 20052.602} C_VEL
LIN {X 0,Y 434.795,Z 807.228,A -85,B 0,C 180,E1 20050.243,E2 20050.243} C_VEL
LIN {X 0,Y 436.125,Z 792.314,A -85,B 0,C 180,E1 20047.915,E2 20047.915} C_VEL
LIN {X 0,Y 437.756,Z 775.626,A -85,B 0,C 180,E1 20045.725,E2 20045.725} C_VEL
LIN {X 0,Y 439.603,Z 757.758,A -85,B 0,C 180,E1 20043.756,E2 20043.756} C_VEL
LIN {X 0,Y 441.51,Z 739.029,A -85,B 0,C 180,E1 20042.031,E2 20042.031} C_VEL
LIN {X 0,Y 443.451,Z 719.67,A -85,B 0,C 180,E1 20040.56,E2 20040.56} C_VEL
LIN {X 0,Y 445.278,Z 700.21,A -85,B 0,C 180,E1 20039.356,E2 20039.356} C_VEL
LIN {X 0,Y 446.967,Z 679.972,A -85,B 0,C 180,E1 20038.361,E2 20038.361} C_VEL
LIN {X 0,Y 448.497,Z 659.076,A -85,B 0,C 180,E1 20037.593,E2 20037.593} C_VEL
LIN {X 0,Y 449.61,Z 636.961,A -85,B 0,C 180,E1 20037.03,E2 20037.03} C_VEL
LIN {X 0,Y 454.893,Z 415.646,A -85,B 0,C 180,E1 20033.089,E2 20033.089} C_VEL
LIN {X 0,Y 451.359,Z 384.026,A -85,B 0,C 180,E1 20032.15,E2 20032.15} C_VEL
LIN {X 0,Y 453.541,Z 356.253,A -85,B 0,C 180,E1 20030.096,E2 20030.096} C_VEL
LIN {X 0,Y 445.35,Z 335.77,A -85,B 0,C 180,E1 20027.615,E2 20027.615} C_VEL
LIN {X 0,Y 437.614,Z 318.561,A -85,B 0,C 180,E1 20025.281,E2 20025.281} C_VEL
LIN {X 0,Y 434.4,Z 311.792,A -85,B 0,C 180,E1 20024.291,E2 20024.291} C_VEL
LIN {X 0,Y 433.262,Z 308.771,A -85,B 0,C 180,E1 20023.814,E2 20023.814} C_VEL
LIN {X 0,Y 433.249,Z 308.485,A -85,B 0,C 180,E1 20020.602,E2 20020.602} C_VEL
LIN {X 0,Y 433.256,Z 308.473,A -85,B 0,C 180,E1 20016.871,E2 20016.871} C_VEL
LIN {X 0,Y 433.256,Z 308.517,A -85,B 0,C 180,E1 20012.999,E2 20012.999} C_VEL
LIN {X 0,Y 433.232,Z 308.521,A -85,B 0,C 180,E1 20009.266,E2 20009.266} C_VEL
LIN {X 0,Y 433.213,Z 308.522,A -85,B 0,C 180,E1 20005.524,E2 20005.524} C_VEL
LIN {X 0,Y 433.205,Z 308.52,A -85,B 0,C 180,E1 20001.814,E2 20001.814} C_VEL
LIN {X 0,Y 433.215,Z 308.507,A -85,B 0,C 180,E1 19998.154,E2 19998.154} C_VEL
LIN {X 0,Y 433.237,Z 308.504,A -85,B 0,C 180,E1 19994.433,E2 19994.433} C_VEL
LIN {X 0,Y 433.241,Z 308.521,A -85,B 0,C 180,E1 19990.639,E2 19990.639} C_VEL
LIN {X 0,Y 433.218,Z 308.511,A -85,B 0,C 180,E1 19986.893,E2 19986.893} C_VEL
LIN {X 0,Y 433.192,Z 308.507,A -85,B 0,C 180,E1 19983.175,E2 19983.175} C_VEL
LIN {X 0,Y 433.181,Z 308.524,A -85,B 0,C 180,E1 19979.471,E2 19979.471} C_VEL
LIN {X 0,Y 433.182,Z 308.52,A -85,B 0,C 180,E1 19975.631,E2 19975.631} C_VEL
LIN {X 0,Y 433.201,Z 308.502,A -85,B 0,C 180,E1 19971.945,E2 19971.945} C_VEL
LIN {X 0,Y 433.236,Z 308.52,A -85,B 0,C 180,E1 19968.282,E2 19968.282} C_VEL
LIN {X 0,Y 433.239,Z 308.506,A -85,B 0,C 180,E1 19964.472,E2 19964.472} C_VEL
LIN {X 0,Y 433.215,Z 308.505,A -85,B 0,C 180,E1 19960.725,E2 19960.725} C_VEL
LIN {X 0,Y 433.203,Z 308.522,A -85,B 0,C 180,E1 19957.041,E2 19957.041} C_VEL
LIN {X 0,Y 433.204,Z 308.521,A -85,B 0,C 180,E1 19953.251,E2 19953.251} C_VEL
LIN {X 0,Y 433.214,Z 308.515,A -85,B 0,C 180,E1 19949.485,E2 19949.485} C_VEL
LIN {X 0,Y 433.246,Z 308.506,A -85,B 0,C 180,E1 19945.888,E2 19945.888} C_VEL
LIN {X 0,Y 433.261,Z 308.506,A -85,B 0,C 180,E1 19942.113,E2 19942.113} C_VEL
LIN {X 0,Y 433.247,Z 308.508,A -85,B 0,C 180,E1 19938.344,E2 19938.344} C_VEL
LIN {X 0,Y 433.23,Z 308.48,A -85,B 0,C 180,E1 19934.554,E2 19934.554} C_VEL
LIN {X 0,Y 433.224,Z 308.523,A -85,B 0,C 180,E1 19930.778,E2 19930.778} C_VEL
LIN {X 0,Y 433.288,Z 308.703,A -85,B 0,C 180,E1 19927.865,E2 19927.865} C_VEL
LIN {X 0,Y 439.62,Z 325.147,A -85,B 0,C 180,E1 19924.968,E2 19924.968} C_VEL
LIN {X 0,Y 445.697,Z 342.303,A -85,B 0,C 180,E1 19922.308,E2 19922.308} C_VEL
LIN {X 0,Y 451.327,Z 353.188,A -85,B 0,C 180,E1 19921.59,E2 19921.59} C_VEL
LIN {X 0,Y 453.612,Z 365.256,A -85,B 0,C 180,E1 19921.173,E2 19921.173} C_VEL
LIN {X 0,Y 451.164,Z 520.038,A -85,B 0,C 180,E1 19918.752,E2 19918.752} C_VEL
LIN {X 0,Y 450.198,Z 527.737,A -85,B 0,C 180,E1 19918.703,E2 19918.703} C_VEL
LIN {X 0,Y 444.61,Z 548.211,A -85,B 0,C 180,E1 19918.805,E2 19918.805} C_VEL
LIN {X 0,Y 443.897,Z 554.794,A -85,B 0,C 180,E1 19918.73,E2 19918.73} C_VEL
LIN {X 0,Y 443.414,Z 573.367,A -85,B 0,C 180,E1 19918.233,E2 19918.233} C_VEL
LIN {X 0,Y 442.477,Z 591.376,A -85,B 0,C 180,E1 19917.522,E2 19917.522} C_VEL
LIN {X 0,Y 441.192,Z 608.876,A -85,B 0,C 180,E1 19916.588,E2 19916.588} C_VEL
LIN {X 0,Y 439.554,Z 625.744,A -85,B 0,C 180,E1 19915.436,E2 19915.436} C_VEL
LIN {X 0,Y 437.703,Z 641.812,A -85,B 0,C 180,E1 19914.063,E2 19914.063} C_VEL
LIN {X 0,Y 435.672,Z 657.035,A -85,B 0,C 180,E1 19912.464,E2 19912.464} C_VEL
LIN {X 0,Y 433.613,Z 671.113,A -85,B 0,C 180,E1 19910.658,E2 19910.658} C_VEL
LIN {X 0,Y 431.721,Z 683.211,A -85,B 0,C 180,E1 19908.779,E2 19908.779} C_VEL
LIN {X 0,Y 429.901,Z 694.651,A -85,B 0,C 180,E1 19906.619,E2 19906.619} C_VEL
LIN {X 0,Y 428.36,Z 704.508,A -85,B 0,C 180,E1 19904.325,E2 19904.325} C_VEL
LIN {X 0,Y 427.097,Z 712.854,A -85,B 0,C 180,E1 19901.888,E2 19901.888} C_VEL
LIN {X 0,Y 426.22,Z 719.323,A -85,B 0,C 180,E1 19899.451,E2 19899.451} C_VEL
LIN {X 0,Y 425.589,Z 724.368,A -85,B 0,C 180,E1 19896.881,E2 19896.881} C_VEL
LIN {X 0,Y 425.222,Z 727.728,A -85,B 0,C 180,E1 19894.315,E2 19894.315} C_VEL
LIN {X 0,Y 425.048,Z 729.585,A -85,B 0,C 180,E1 19891.618,E2 19891.618} C_VEL
LIN {X 0,Y 425.026,Z 729.784,A -85,B 0,C 180,E1 19888.922,E2 19888.922} C_VEL
LIN {X 0,Y 425.165,Z 728.333,A -85,B 0,C 180,E1 19886.225,E2 19886.225} C_VEL
LIN {X 0,Y 425.506,Z 725.175,A -85,B 0,C 180,E1 19883.524,E2 19883.524} C_VEL
LIN {X 0,Y 426.124,Z 720.184,A -85,B 0,C 180,E1 19880.819,E2 19880.819} C_VEL
LIN {X 0,Y 427.01,Z 713.565,A -85,B 0,C 180,E1 19878.246,E2 19878.246} C_VEL
LIN {X 0,Y 428.236,Z 705.404,A -85,B 0,C 180,E1 19875.809,E2 19875.809} C_VEL
LIN {X 0,Y 429.75,Z 695.733,A -85,B 0,C 180,E1 19873.511,E2 19873.511} C_VEL
LIN {X 0,Y 431.529,Z 684.545,A -85,B 0,C 180,E1 19871.353,E2 19871.353} C_VEL
LIN {X 0,Y 433.398,Z 672.724,A -85,B 0,C 180,E1 19869.473,E2 19869.473} C_VEL
LIN {X 0,Y 435.425,Z 658.978,A -85,B 0,C 180,E1 19867.665,E2 19867.665} C_VEL
LIN {X 0,Y 437.429,Z 644.175,A -85,B 0,C 180,E1 19866.064,E2 19866.064} C_VEL
LIN {X 0,Y 439.316,Z 628.345,A -85,B 0,C 180,E1 19864.668,E2 19864.668} C_VEL
LIN {X 0,Y 441.008,Z 611.462,A -85,B 0,C 180,E1 19863.472,E2 19863.472} C_VEL
LIN {X 0,Y 442.353,Z 594.052,A -85,B 0,C 180,E1 19862.506,E2 19862.506} C_VEL
LIN {X 0,Y 443.357,Z 575.671,A -85,B 0,C 180,E1 19861.747,E2 19861.747} C_VEL
LIN {X 0,Y 443.911,Z 556.954,A -85,B 0,C 180,E1 19861.219,E2 19861.219} C_VEL
LIN {X 0,Y 446.899,Z 364.901,A -85,B 0,C 180,E1 19858.123,E2 19858.123} C_VEL
LIN {X 0,Y 444.689,Z 355.34,A -85,B 0,C 180,E1 19857.747,E2 19857.747} C_VEL
LIN {X 0,Y 437.741,Z 342.648,A -85,B 0,C 180,E1 19856.839,E2 19856.839} C_VEL
LIN {X 0,Y 431.644,Z 325.832,A -85,B 0,C 180,E1 19854.124,E2 19854.124} C_VEL
LIN {X 0,Y 426.384,Z 312.582,A -85,B 0,C 180,E1 19851.753,E2 19851.753} C_VEL
LIN {X 0,Y 425.328,Z 309.748,A -85,B 0,C 180,E1 19851.195,E2 19851.195} C_VEL
LIN {X 0,Y 425.313,Z 309.498,A -85,B 0,C 180,E1 19848.382,E2 19848.382} C_VEL
LIN {X 0,Y 425.295,Z 309.481,A -85,B 0,C 180,E1 19844.576,E2 19844.576} C_VEL
LIN {X 0,Y 425.284,Z 309.502,A -85,B 0,C 180,E1 19840.799,E2 19840.799} C_VEL
LIN {X 0,Y 425.28,Z 309.504,A -85,B 0,C 180,E1 19836.933,E2 19836.933} C_VEL
LIN {X 0,Y 425.281,Z 309.5,A -85,B 0,C 180,E1 19833.181,E2 19833.181} C_VEL
LIN {X 0,Y 425.298,Z 309.492,A -85,B 0,C 180,E1 19829.43,E2 19829.43} C_VEL
LIN {X 0,Y 425.31,Z 309.492,A -85,B 0,C 180,E1 19825.631,E2 19825.631} C_VEL
LIN {X 0,Y 425.32,Z 309.507,A -85,B 0,C 180,E1 19821.79,E2 19821.79} C_VEL
LIN {X 0,Y 425.296,Z 309.501,A -85,B 0,C 180,E1 19817.938,E2 19817.938} C_VEL
LIN {X 0,Y 425.262,Z 309.49,A -85,B 0,C 180,E1 19814.293,E2 19814.293} C_VEL
LIN {X 0,Y 425.254,Z 309.509,A -85,B 0,C 180,E1 19810.568,E2 19810.568} C_VEL
LIN {X 0,Y 425.25,Z 309.511,A -85,B 0,C 180,E1 19806.752,E2 19806.752} C_VEL
LIN {X 0,Y 425.262,Z 309.489,A -85,B 0,C 180,E1 19803.1,E2 19803.1} C_VEL
LIN {X 0,Y 425.286,Z 309.505,A -85,B 0,C 180,E1 19799.327,E2 19799.327} C_VEL
LIN {X 0,Y 425.292,Z 309.502,A -85,B 0,C 180,E1 19795.409,E2 19795.409} C_VEL
LIN {X 0,Y 425.286,Z 309.489,A -85,B 0,C 180,E1 19791.619,E2 19791.619} C_VEL
LIN {X 0,Y 425.266,Z 309.506,A -85,B 0,C 180,E1 19787.922,E2 19787.922} C_VEL
LIN {X 0,Y 425.258,Z 309.511,A -85,B 0,C 180,E1 19784.313,E2 19784.313} C_VEL
LIN {X 0,Y 425.265,Z 309.505,A -85,B 0,C 180,E1 19780.497,E2 19780.497} C_VEL
LIN {X 0,Y 425.282,Z 309.495,A -85,B 0,C 180,E1 19776.736,E2 19776.736} C_VEL
LIN {X 0,Y 425.308,Z 309.493,A -85,B 0,C 180,E1 19772.995,E2 19772.995} C_VEL
LIN {X 0,Y 425.323,Z 309.493,A -85,B 0,C 180,E1 19769.171,E2 19769.171} C_VEL
LIN {X 0,Y 425.308,Z 309.471,A -85,B 0,C 180,E1 19765.325,E2 19765.325} C_VEL
LIN {X 0,Y 425.306,Z 309.504,A -85,B 0,C 180,E1 19761.465,E2 19761.465} C_VEL
LIN {X 0,Y 425.285,Z 309.467,A -85,B 0,C 180,E1 19757.748,E2 19757.748} C_VEL
LIN {X 0,Y 425.365,Z 309.797,A -85,B 0,C 180,E1 19757.072,E2 19757.072} C_VEL
LIN {X 0,Y 426.875,Z 313.366,A -85,B 0,C 180,E1 19756.479,E2 19756.479} C_VEL
LIN {X 0,Y 435.021,Z 330.98,A -85,B 0,C 180,E1 19753.9,E2 19753.9} C_VEL
LIN {X 0,Y 442.907,Z 349.683,A -85,B 0,C 180,E1 19751.454,E2 19751.454} C_VEL
LIN {X 0,Y 446.657,Z 359.89,A -85,B 0,C 180,E1 19750.241,E2 19750.241} C_VEL
LIN {X 0,Y 444.624,Z 384.536,A -85,B 0,C 180,E1 19748.424,E2 19748.424} C_VEL
LIN {X 0,Y 448.182,Z 418.162,A -85,B 0,C 180,E1 19747.434,E2 19747.434} C_VEL
LIN {X 0,Y 442.654,Z 636.743,A -85,B 0,C 180,E1 19743.483,E2 19743.483} C_VEL
LIN {X 0,Y 441.487,Z 658.553,A -85,B 0,C 180,E1 19742.914,E2 19742.914} C_VEL
LIN {X 0,Y 439.862,Z 679.388,A -85,B 0,C 180,E1 19742.133,E2 19742.133} C_VEL
LIN {X 0,Y 438.112,Z 699.129,A -85,B 0,C 180,E1 19741.149,E2 19741.149} C_VEL
LIN {X 0,Y 436.149,Z 718.774,A -85,B 0,C 180,E1 19739.915,E2 19739.915} C_VEL
LIN {X 0,Y 434.065,Z 738.298,A -85,B 0,C 180,E1 19738.402,E2 19738.402} C_VEL
LIN {X 0,Y 432.059,Z 756.705,A -85,B 0,C 180,E1 19736.675,E2 19736.675} C_VEL
LIN {X 0,Y 430.138,Z 774.036,A -85,B 0,C 180,E1 19734.734,E2 19734.734} C_VEL
LIN {X 0,Y 428.44,Z 790.259,A -85,B 0,C 180,E1 19732.575,E2 19732.575} C_VEL
LIN {X 0,Y 427.035,Z 804.845,A -85,B 0,C 180,E1 19730.274,E2 19730.274} C_VEL
LIN {X 0,Y 425.959,Z 817.51,A -85,B 0,C 180,E1 19727.908,E2 19727.908} C_VEL
LIN {X 0,Y 425.186,Z 828.803,A -85,B 0,C 180,E1 19725.39,E2 19725.39} C_VEL
LIN {X 0,Y 424.667,Z 838.385,A -85,B 0,C 180,E1 19722.786,E2 19722.786} C_VEL
LIN {X 0,Y 424.416,Z 845.701,A -85,B 0,C 180,E1 19720.314,E2 19720.314} C_VEL
LIN {X 0,Y 424.309,Z 851.575,A -85,B 0,C 180,E1 19717.719,E2 19717.719} C_VEL
LIN {X 0,Y 424.311,Z 855.65,A -85,B 0,C 180,E1 19715.137,E2 19715.137} C_VEL
LIN {X 0,Y 424.338,Z 858.142,A -85,B 0,C 180,E1 19712.488,E2 19712.488} C_VEL
LIN {X 0,Y 424.358,Z 858.961,A -85,B 0,C 180,E1 19710,E2 19710} C_VEL
LIN {X 0,Y 424.339,Z 858.102,A -85,B 0,C 180,E1 19707.434,E2 19707.434} C_VEL
LIN {X 0,Y 424.311,Z 855.659,A -85,B 0,C 180,E1 19704.863,E2 19704.863} C_VEL
LIN {X 0,Y 424.308,Z 851.579,A -85,B 0,C 180,E1 19702.281,E2 19702.281} C_VEL
LIN {X 0,Y 424.417,Z 845.711,A -85,B 0,C 180,E1 19699.686,E2 19699.686} C_VEL
LIN {X 0,Y 424.667,Z 838.393,A -85,B 0,C 180,E1 19697.214,E2 19697.214} C_VEL
LIN {X 0,Y 425.192,Z 828.726,A -85,B 0,C 180,E1 19694.59,E2 19694.59} C_VEL
LIN {X 0,Y 425.959,Z 817.513,A -85,B 0,C 180,E1 19692.092,E2 19692.092} C_VEL
LIN {X 0,Y 427.036,Z 804.848,A -85,B 0,C 180,E1 19689.726,E2 19689.726} C_VEL
LIN {X 0,Y 428.441,Z 790.258,A -85,B 0,C 180,E1 19687.425,E2 19687.425} C_VEL
LIN {X 0,Y 430.138,Z 774.029,A -85,B 0,C 180,E1 19685.266,E2 19685.266} C_VEL
LIN {X 0,Y 432.059,Z 756.695,A -85,B 0,C 180,E1 19683.325,E2 19683.325} C_VEL
LIN {X 0,Y 434.064,Z 738.281,A -85,B 0,C 180,E1 19681.598,E2 19681.598} C_VEL
LIN {X 0,Y 436.146,Z 718.743,A -85,B 0,C 180,E1 19680.085,E2 19680.085} C_VEL
LIN {X 0,Y 438.106,Z 699.108,A -85,B 0,C 180,E1 19678.852,E2 19678.852} C_VEL
LIN {X 0,Y 439.858,Z 679.336,A -85,B 0,C 180,E1 19677.866,E2 19677.866} C_VEL
LIN {X 0,Y 441.493,Z 658.348,A -85,B 0,C 180,E1 19677.081,E2 19677.081} C_VEL
LIN {X 0,Y 442.667,Z 636.086,A -85,B 0,C 180,E1 19676.506,E2 19676.506} C_VEL
LIN {X 0,Y 448.204,Z 416.738,A -85,B 0,C 180,E1 19672.543,E2 19672.543} C_VEL
LIN {X 0,Y 444.573,Z 383.333,A -85,B 0,C 180,E1 19671.523,E2 19671.523} C_VEL
LIN {X 0,Y 446.59,Z 359.288,A -85,B 0,C 180,E1 19669.709,E2 19669.709} C_VEL
LIN {X 0,Y 438.573,Z 339.092,A -85,B 0,C 180,E1 19667.206,E2 19667.206} C_VEL
LIN {X 0,Y 430.583,Z 321.167,A -85,B 0,C 180,E1 19664.716,E2 19664.716} C_VEL
LIN {X 0,Y 425.441,Z 310.203,A -85,B 0,C 180,E1 19663.04,E2 19663.04} C_VEL
LIN {X 0,Y 425.323,Z 309.528,A -85,B 0,C 180,E1 19662.796,E2 19662.796} C_VEL
LIN {X 0,Y 425.328,Z 309.508,A -85,B 0,C 180,E1 19658.914,E2 19658.914} C_VEL
LIN {X 0,Y 425.312,Z 309.465,A -85,B 0,C 180,E1 19655.002,E2 19655.002} C_VEL
LIN {X 0,Y 425.293,Z 309.498,A -85,B 0,C 180,E1 19651.303,E2 19651.303} C_VEL
LIN {X 0,Y 425.275,Z 309.499,A -85,B 0,C 180,E1 19647.584,E2 19647.584} C_VEL
LIN {X 0,Y 425.269,Z 309.503,A -85,B 0,C 180,E1 19643.853,E2 19643.853} C_VEL
LIN {X 0,Y 425.274,Z 309.507,A -85,B 0,C 180,E1 19640.075,E2 19640.075} C_VEL
LIN {X 0,Y 425.295,Z 309.51,A -85,B 0,C 180,E1 19636.386,E2 19636.386} C_VEL
LIN {X 0,Y 425.304,Z 309.491,A -85,B 0,C 180,E1 19632.629,E2 19632.629} C_VEL
LIN {X 0,Y 425.291,Z 309.491,A -85,B 0,C 180,E1 19628.79,E2 19628.79} C_VEL
LIN {X 0,Y 425.259,Z 309.512,A -85,B 0,C 180,E1 19625.126,E2 19625.126} C_VEL
LIN {X 0,Y 425.246,Z 309.506,A -85,B 0,C 180,E1 19621.347,E2 19621.347} C_VEL
LIN {X 0,Y 425.238,Z 309.495,A -85,B 0,C 180,E1 19617.574,E2 19617.574} C_VEL
LIN {X 0,Y 425.253,Z 309.511,A -85,B 0,C 180,E1 19613.791,E2 19613.791} C_VEL
LIN {X 0,Y 425.279,Z 309.498,A -85,B 0,C 180,E1 19610.086,E2 19610.086} C_VEL
LIN {X 0,Y 425.305,Z 309.487,A -85,B 0,C 180,E1 19606.264,E2 19606.264} C_VEL
LIN {X 0,Y 425.294,Z 309.508,A -85,B 0,C 180,E1 19602.486,E2 19602.486} C_VEL
LIN {X 0,Y 425.275,Z 309.503,A -85,B 0,C 180,E1 19598.772,E2 19598.772} C_VEL
LIN {X 0,Y 425.262,Z 309.492,A -85,B 0,C 180,E1 19595.111,E2 19595.111} C_VEL
LIN {X 0,Y 425.268,Z 309.502,A -85,B 0,C 180,E1 19591.276,E2 19591.276} C_VEL
LIN {X 0,Y 425.284,Z 309.507,A -85,B 0,C 180,E1 19587.565,E2 19587.565} C_VEL
LIN {X 0,Y 425.308,Z 309.508,A -85,B 0,C 180,E1 19583.837,E2 19583.837} C_VEL
LIN {X 0,Y 425.328,Z 309.506,A -85,B 0,C 180,E1 19580.026,E2 19580.026} C_VEL
LIN {X 0,Y 425.318,Z 309.499,A -85,B 0,C 180,E1 19576.092,E2 19576.092} C_VEL
LIN {X 0,Y 425.311,Z 309.478,A -85,B 0,C 180,E1 19572.223,E2 19572.223} C_VEL
LIN {X 0,Y 425.322,Z 309.731,A -85,B 0,C 180,E1 19568.704,E2 19568.704} C_VEL
LIN {X 0,Y 431.316,Z 325.075,A -85,B 0,C 180,E1 19565.907,E2 19565.907} C_VEL
LIN {X 0,Y 437.334,Z 341.625,A -85,B 0,C 180,E1 19563.199,E2 19563.199} C_VEL
LIN {X 0,Y 438.46,Z 344.163,A -85,B 0,C 180,E1 19562.946,E2 19562.946} C_VEL
LIN {X 0,Y 445.18,Z 356.721,A -85,B 0,C 180,E1 19562.081,E2 19562.081} C_VEL
LIN {X 0,Y 447.01,Z 366.68,A -85,B 0,C 180,E1 19561.733,E2 19561.733} C_VEL
LIN {X 0,Y 443.897,Z 554.794,A -85,B 0,C 180,E1 19558.73,E2 19558.73} C_VEL
LIN {X 0,Y 442.939,Z 562.472,A -85,B 0,C 180,E1 19558.628,E2 19558.628} C_VEL
LIN {X 0,Y 437.427,Z 580.609,A -85,B 0,C 180,E1 19558.46,E2 19558.46} C_VEL
LIN {X 0,Y 435.926,Z 588.027,A -85,B 0,C 180,E1 19558.239,E2 19558.239} C_VEL
LIN {X 0,Y 435.833,Z 589.062,A -85,B 0,C 180,E1 19558.193,E2 19558.193} C_VEL
LIN {X 0,Y 434.586,Z 606.139,A -85,B 0,C 180,E1 19557.321,E2 19557.321} C_VEL
